// TIA Portal V17 export
// export: Created 2024-09-02T12:50:15.2949432Z, ExportSetting WithDefaults, DisplayName Totally Integrated Automation Portal, DisplayVersion V17, DisplayName TIA Portal Openness, DisplayVersion V17, DisplayName TIA Portal Version Control Interface, DisplayVersion V17, DisplayName STEP 7 Professional, DisplayVersion V17, DisplayName STEP 7 Safety, DisplayVersion V17, DisplayName WinCC Professional, DisplayVersion V17
FUNCTION "AnwFC_ZP_Alarm_OP70" : Void   // FC155, LAD
TITLE = Störmeldungen und Betriebsmeldungen rangieren
{ S7_Optimized_Access := 'TRUE' }
AUTHOR : OlegFuehrus
FAMILY : BA
NAME : BA
VERSION : 0.1
// stored: AutoNumber true, IsIECCheckEnabled false, SetENOAutomatically false, UDAEnableTagReadback false
   VAR_TEMP
      t_bTemp : Bool;
      t_ControlVoltage : Bool;
      t_StartReady : Bool;
      t_OverviewStartCon : Bool;
      t_EStop_NOK : Bool;
      t_Fault : Bool;
      t_oppen_SG : Array[1..8] of Bool;
      t_wert : Byte;
      t_status : Word;
      t_RetValSFC : Int;
      _NumOf_ParFlt_General : Int;
      _NumOf_SQFlt_General : Int;
      _NumOf_Flt_General_A : Int;
      _NumOf_Flt_General_B : Int;
      _NumOf_Flt_SubSys : Int;
      _NumOf_Reports : Int;
      _NumOf_Rep : Int;
   END_VAR
   VAR_TEMP   // added for the SCL form of the ladder/FBD networks
      _w1 : Bool;
      _w2 : Bool;
      _w3 : Bool;
      _w4 : Bool;
      _w5 : Bool;
   END_VAR
BEGIN

REGION Network 1: INIT
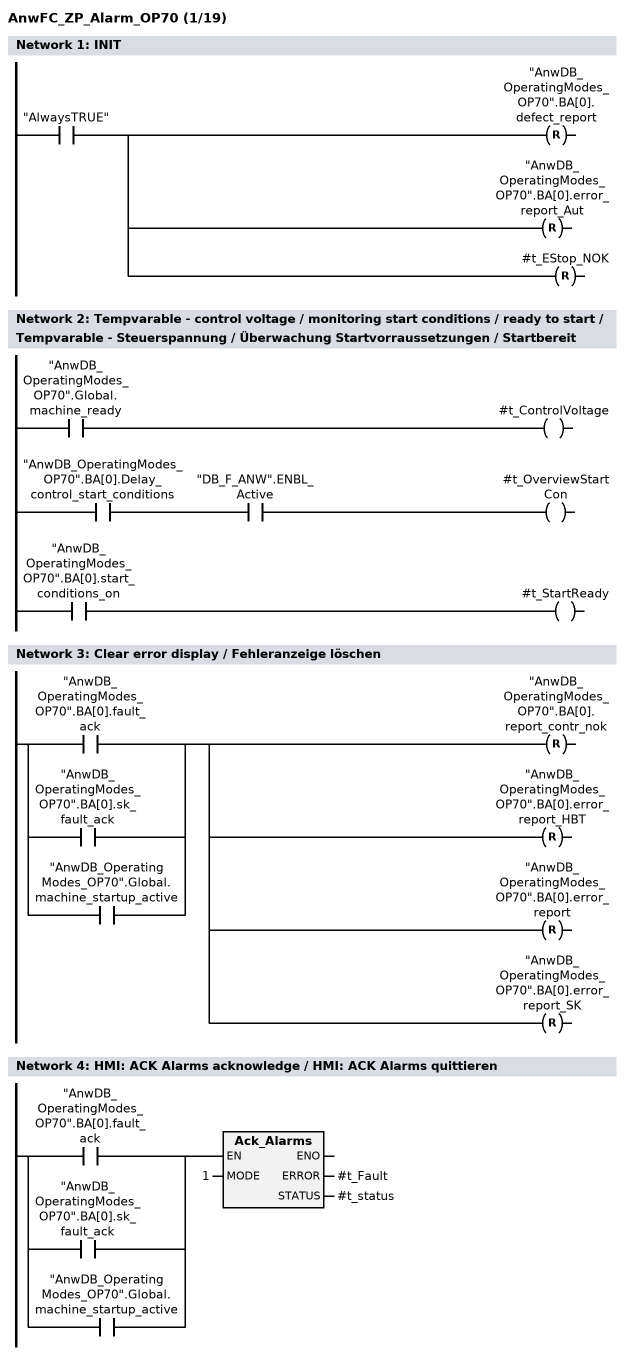
   RUNG wire#powerrail
      Contact( "AlwaysTRUE" )
      wire#w1
      R_Coil( "AnwDB_OperatingModes_OP70".BA[0].defect_report )
   END_RUNG
   RUNG wire#w1
      R_Coil( "AnwDB_OperatingModes_OP70".BA[0].error_report_Aut )
   END_RUNG
   RUNG wire#w1
      R_Coil( #t_EStop_NOK )
   END_RUNG
   // the same network as SCL:
   IF "AlwaysTRUE" THEN
       "AnwDB_OperatingModes_OP70".BA[0].defect_report := FALSE;
       "AnwDB_OperatingModes_OP70".BA[0].error_report_Aut := FALSE;
       #t_EStop_NOK := FALSE;
   END_IF;
END_REGION

REGION Network 2: Tempvarable - control voltage / monitoring start conditions / ready to start / Tempvarable - Steuerspannung / Überwachung Startvorraussetzungen / Startbereit
   RUNG wire#powerrail
      Contact( "AnwDB_OperatingModes_OP70".Global.machine_ready )
      Coil( #t_ControlVoltage )
   END_RUNG
   RUNG wire#powerrail
      Contact( "AnwDB_OperatingModes_OP70".BA[0].Delay_control_start_conditions )
      Contact( "DB_F_ANW".ENBL_Active )
      Coil( #t_OverviewStartCon )
   END_RUNG
   RUNG wire#powerrail
      Contact( "AnwDB_OperatingModes_OP70".BA[0].start_conditions_on )
      Coil( #t_StartReady )
   END_RUNG
   // the same network as SCL:
   #t_ControlVoltage := "AnwDB_OperatingModes_OP70".Global.machine_ready;
   #t_OverviewStartCon := "AnwDB_OperatingModes_OP70".BA[0].Delay_control_start_conditions AND "DB_F_ANW".ENBL_Active;
   #t_StartReady := "AnwDB_OperatingModes_OP70".BA[0].start_conditions_on;
END_REGION

REGION Network 3: Clear error display / Fehleranzeige löschen
   RUNG wire#powerrail
      Contact( "AnwDB_OperatingModes_OP70".BA[0].fault_ack )
      wire#w1
      R_Coil( "AnwDB_OperatingModes_OP70".BA[0].report_contr_nok )
   END_RUNG
   RUNG wire#powerrail
      Contact( "AnwDB_OperatingModes_OP70".BA[0].sk_fault_ack )
   END_RUNG wire#w1
   RUNG wire#powerrail
      Contact( "AnwDB_OperatingModes_OP70".Global.machine_startup_active )
   END_RUNG wire#w1
   RUNG wire#w1
      R_Coil( "AnwDB_OperatingModes_OP70".BA[0].error_report_HBT )
   END_RUNG
   RUNG wire#w1
      R_Coil( "AnwDB_OperatingModes_OP70".BA[0].error_report )
   END_RUNG
   RUNG wire#w1
      R_Coil( "AnwDB_OperatingModes_OP70".BA[0].error_report_SK )
   END_RUNG
   // the same network as SCL:
   #_w1 := "AnwDB_OperatingModes_OP70".BA[0].fault_ack OR "AnwDB_OperatingModes_OP70".BA[0].sk_fault_ack OR "AnwDB_OperatingModes_OP70".Global.machine_startup_active;
   IF #_w1 THEN
       "AnwDB_OperatingModes_OP70".BA[0].report_contr_nok := FALSE;
       "AnwDB_OperatingModes_OP70".BA[0].error_report_HBT := FALSE;
       "AnwDB_OperatingModes_OP70".BA[0].error_report := FALSE;
       "AnwDB_OperatingModes_OP70".BA[0].error_report_SK := FALSE;
   END_IF;
END_REGION

REGION Network 4: HMI: ACK Alarms acknowledge / HMI: ACK Alarms quittieren
   RUNG wire#powerrail
      Contact( "AnwDB_OperatingModes_OP70".BA[0].fault_ack )
      wire#w1
      Ack_Alarms(MODE := 1, ERROR => #t_Fault, STATUS => #t_status)
   END_RUNG
   RUNG wire#powerrail
      Contact( "AnwDB_OperatingModes_OP70".BA[0].sk_fault_ack )
   END_RUNG wire#w1
   RUNG wire#powerrail
      Contact( "AnwDB_OperatingModes_OP70".Global.machine_startup_active )
   END_RUNG wire#w1
   // the same network as SCL:
   IF "AnwDB_OperatingModes_OP70".BA[0].fault_ack OR "AnwDB_OperatingModes_OP70".BA[0].sk_fault_ack OR "AnwDB_OperatingModes_OP70".Global.machine_startup_active THEN
       Ack_Alarms(MODE := 1, ERROR => #t_Fault, STATUS => #t_status);
   END_IF;
END_REGION

REGION Network 5: Acknowledge fault at MP / Störung am MP quittieren
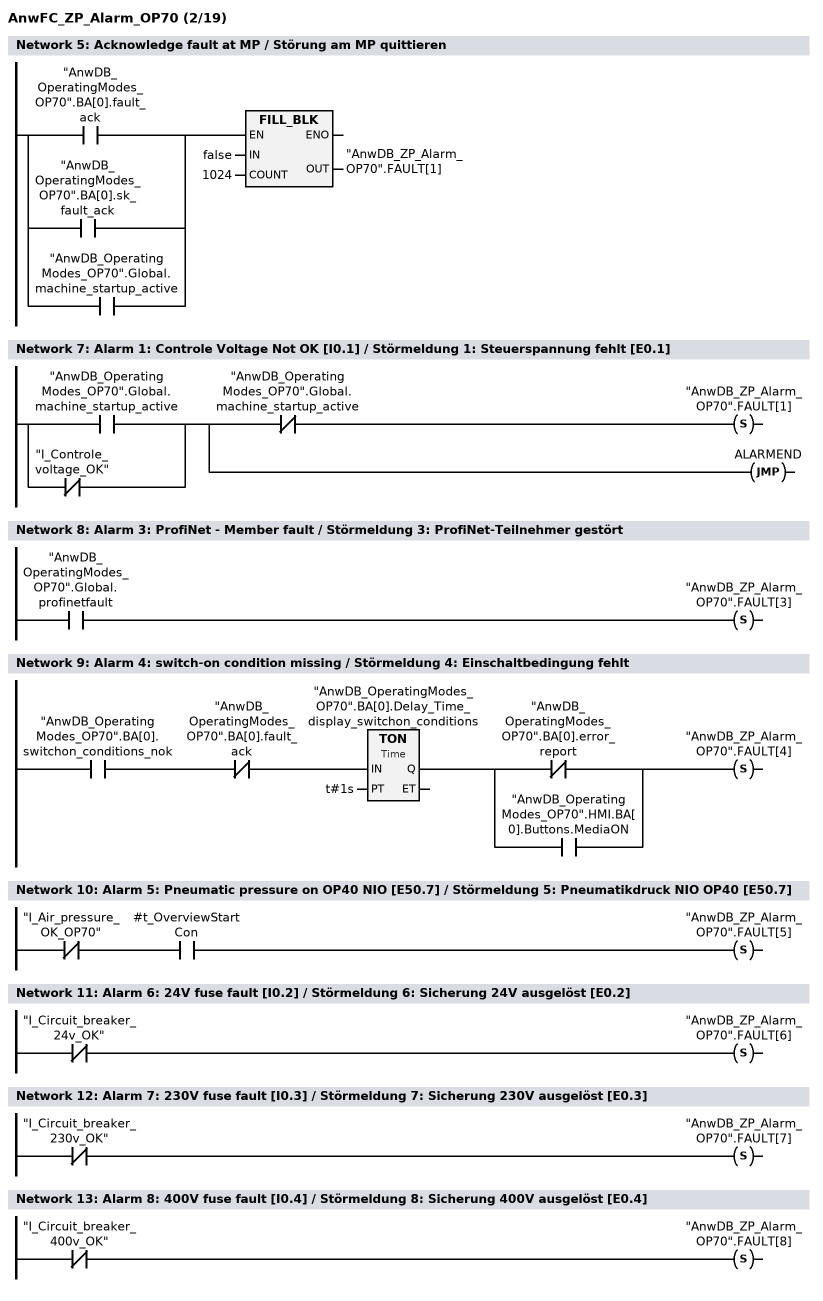
   RUNG wire#powerrail
      Contact( "AnwDB_OperatingModes_OP70".BA[0].fault_ack )
      wire#w1
      FillBlockI(in := false, count := 1024, out => "AnwDB_ZP_Alarm_OP70".FAULT[1])
   END_RUNG
   RUNG wire#powerrail
      Contact( "AnwDB_OperatingModes_OP70".BA[0].sk_fault_ack )
   END_RUNG wire#w1
   RUNG wire#powerrail
      Contact( "AnwDB_OperatingModes_OP70".Global.machine_startup_active )
   END_RUNG wire#w1
   // the same network as SCL:
   IF "AnwDB_OperatingModes_OP70".BA[0].fault_ack OR "AnwDB_OperatingModes_OP70".BA[0].sk_fault_ack OR "AnwDB_OperatingModes_OP70".Global.machine_startup_active THEN
       FILL_BLK(IN := false, COUNT := 1024, OUT => "AnwDB_ZP_Alarm_OP70".FAULT[1]);
   END_IF;
END_REGION

REGION Network 6: ########################### Global Power condition############################### / ########################### Störmeldungen ###############################
END_REGION

REGION Network 7: Alarm 1: Controle Voltage Not OK [I0.1] / Störmeldung 1: Steuerspannung fehlt [E0.1]
   RUNG wire#powerrail
      Contact( "AnwDB_OperatingModes_OP70".Global.machine_startup_active )
      wire#w1
      I_Contact( "AnwDB_OperatingModes_OP70".Global.machine_startup_active )
      S_Coil( "AnwDB_ZP_Alarm_OP70".FAULT[1] )
   END_RUNG
   RUNG wire#powerrail
      I_Contact( "I_Controle_voltage_OK" )
   END_RUNG wire#w1
   RUNG wire#w1
      JumpCoil( ALARMEND )
   END_RUNG
   // the same network as SCL:
   #_w1 := "AnwDB_OperatingModes_OP70".Global.machine_startup_active OR NOT "I_Controle_voltage_OK";
   IF #_w1 AND NOT "AnwDB_OperatingModes_OP70".Global.machine_startup_active THEN
       "AnwDB_ZP_Alarm_OP70".FAULT[1] := TRUE;
   END_IF;
   IF #_w1 THEN GOTO ALARMEND; END_IF;
END_REGION

REGION Network 8: Alarm 3: ProfiNet - Member fault / Störmeldung 3: ProfiNet-Teilnehmer gestört
   RUNG wire#powerrail
      Contact( "AnwDB_OperatingModes_OP70".Global.profinetfault )
      S_Coil( "AnwDB_ZP_Alarm_OP70".FAULT[3] )
   END_RUNG
   // the same network as SCL:
   IF "AnwDB_OperatingModes_OP70".Global.profinetfault THEN "AnwDB_ZP_Alarm_OP70".FAULT[3] := TRUE; END_IF;
END_REGION

REGION Network 9: Alarm 4: switch-on condition missing / Störmeldung 4: Einschaltbedingung fehlt
   RUNG wire#powerrail
      Contact( "AnwDB_OperatingModes_OP70".BA[0].switchon_conditions_nok )
      I_Contact( "AnwDB_OperatingModes_OP70".BA[0].fault_ack )
      { S7_Templates := "time_type := Time" } "AnwDB_OperatingModes_OP70".BA[0].Delay_Time_display_switchon_conditions.TON(pt := t#1s, et =>)
      wire#w1
      I_Contact( "AnwDB_OperatingModes_OP70".BA[0].error_report )
      wire#w2
      S_Coil( "AnwDB_ZP_Alarm_OP70".FAULT[4] )
   END_RUNG
   RUNG wire#w1
      Contact( "AnwDB_OperatingModes_OP70".HMI.BA[0].Buttons.MediaON )
   END_RUNG wire#w2
   // the same network as SCL:
   "AnwDB_OperatingModes_OP70".BA[0].Delay_Time_display_switchon_conditions.TON(IN := "AnwDB_OperatingModes_OP70".BA[0].switchon_conditions_nok AND NOT "AnwDB_OperatingModes_OP70".BA[0].fault_ack,
                           PT := t#1s);
   IF "AnwDB_OperatingModes_OP70".BA[0].Delay_Time_display_switchon_conditions.Q AND (NOT "AnwDB_OperatingModes_OP70".BA[0].error_report OR "AnwDB_OperatingModes_OP70".HMI.BA[0].Buttons.MediaON) THEN
       "AnwDB_ZP_Alarm_OP70".FAULT[4] := TRUE;
   END_IF;
END_REGION

REGION Network 10: Alarm 5: Pneumatic pressure on OP40 NIO [E50.7] / Störmeldung 5: Pneumatikdruck NIO OP40 [E50.7]
   RUNG wire#powerrail
      I_Contact( "I_Air_pressure_OK_OP70" )
      Contact( #t_OverviewStartCon )
      S_Coil( "AnwDB_ZP_Alarm_OP70".FAULT[5] )
   END_RUNG
   // the same network as SCL:
   IF NOT "I_Air_pressure_OK_OP70" AND #t_OverviewStartCon THEN
       "AnwDB_ZP_Alarm_OP70".FAULT[5] := TRUE;
   END_IF;
END_REGION

REGION Network 11: Alarm 6: 24V fuse fault [I0.2] / Störmeldung 6: Sicherung 24V ausgelöst [E0.2]
   RUNG wire#powerrail
      I_Contact( "I_Circuit_breaker_24v_OK" )
      S_Coil( "AnwDB_ZP_Alarm_OP70".FAULT[6] )
   END_RUNG
   // the same network as SCL:
   IF NOT "I_Circuit_breaker_24v_OK" THEN "AnwDB_ZP_Alarm_OP70".FAULT[6] := TRUE; END_IF;
END_REGION

REGION Network 12: Alarm 7: 230V fuse fault [I0.3] / Störmeldung 7: Sicherung 230V ausgelöst [E0.3]
   RUNG wire#powerrail
      I_Contact( "I_Circuit_breaker_230v_OK" )
      S_Coil( "AnwDB_ZP_Alarm_OP70".FAULT[7] )
   END_RUNG
   // the same network as SCL:
   IF NOT "I_Circuit_breaker_230v_OK" THEN "AnwDB_ZP_Alarm_OP70".FAULT[7] := TRUE; END_IF;
END_REGION

REGION Network 13: Alarm 8: 400V fuse fault [I0.4] / Störmeldung 8: Sicherung 400V ausgelöst [E0.4]
   RUNG wire#powerrail
      I_Contact( "I_Circuit_breaker_400v_OK" )
      S_Coil( "AnwDB_ZP_Alarm_OP70".FAULT[8] )
   END_RUNG
   // the same network as SCL:
   IF NOT "I_Circuit_breaker_400v_OK" THEN "AnwDB_ZP_Alarm_OP70".FAULT[8] := TRUE; END_IF;
END_REGION

REGION Network 14: Power Condition: ENDE ########################## / ESB: ENDE ##########################
END_REGION

REGION Network 15: Alarm 25: Reworking in Station / Störmeldung 25: Nacharbeit in Station
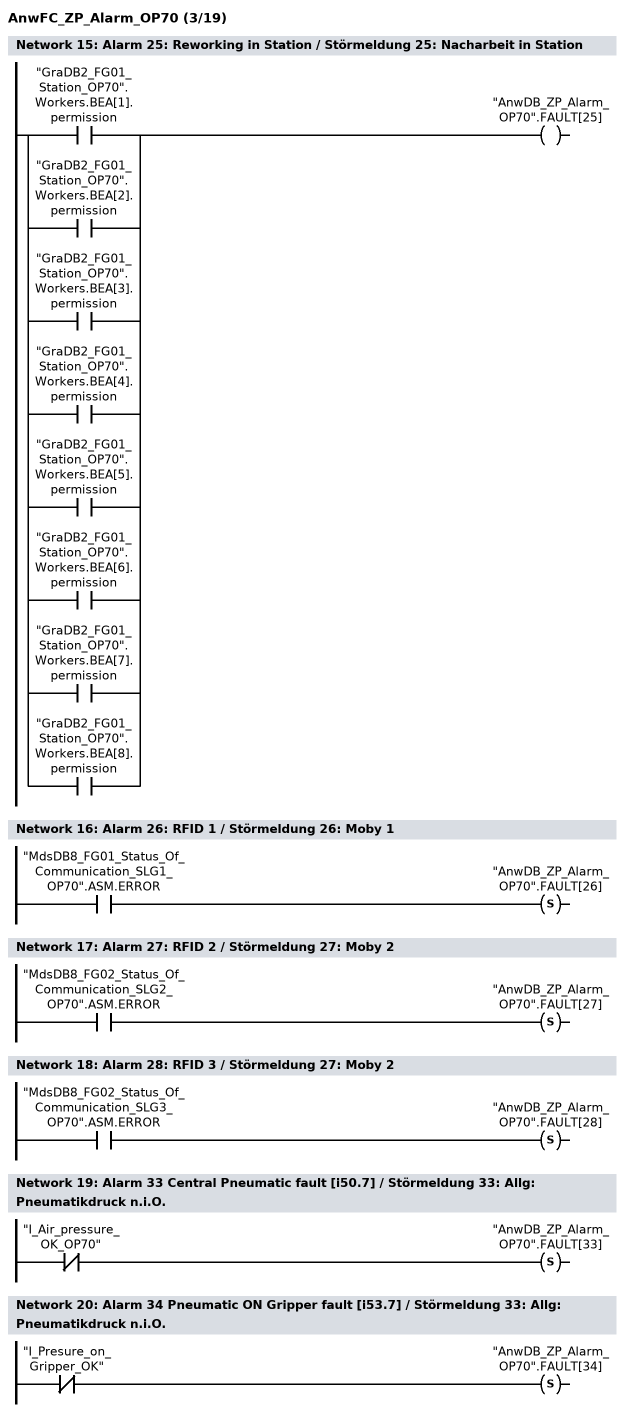
   RUNG wire#powerrail
      Contact( "GraDB2_FG01_Station_OP70".Workers.BEA[1].permission )
      wire#w1
      Coil( "AnwDB_ZP_Alarm_OP70".FAULT[25] )
   END_RUNG
   RUNG wire#powerrail
      Contact( "GraDB2_FG01_Station_OP70".Workers.BEA[2].permission )
   END_RUNG wire#w1
   RUNG wire#powerrail
      Contact( "GraDB2_FG01_Station_OP70".Workers.BEA[3].permission )
   END_RUNG wire#w1
   RUNG wire#powerrail
      Contact( "GraDB2_FG01_Station_OP70".Workers.BEA[4].permission )
   END_RUNG wire#w1
   RUNG wire#powerrail
      Contact( "GraDB2_FG01_Station_OP70".Workers.BEA[5].permission )
   END_RUNG wire#w1
   RUNG wire#powerrail
      Contact( "GraDB2_FG01_Station_OP70".Workers.BEA[6].permission )
   END_RUNG wire#w1
   RUNG wire#powerrail
      Contact( "GraDB2_FG01_Station_OP70".Workers.BEA[7].permission )
   END_RUNG wire#w1
   RUNG wire#powerrail
      Contact( "GraDB2_FG01_Station_OP70".Workers.BEA[8].permission )
   END_RUNG wire#w1
   // the same network as SCL:
   "AnwDB_ZP_Alarm_OP70".FAULT[25] := "GraDB2_FG01_Station_OP70".Workers.BEA[1].permission OR "GraDB2_FG01_Station_OP70".Workers.BEA[2].permission OR "GraDB2_FG01_Station_OP70".Workers.BEA[3].permission OR "GraDB2_FG01_Station_OP70".Workers.BEA[4].permission OR "GraDB2_FG01_Station_OP70".Workers.BEA[5].permission OR "GraDB2_FG01_Station_OP70".Workers.BEA[6].permission OR "GraDB2_FG01_Station_OP70".Workers.BEA[7].permission OR "GraDB2_FG01_Station_OP70".Workers.BEA[8].permission;
END_REGION

REGION Network 16: Alarm 26: RFID 1 / Störmeldung 26: Moby 1
   RUNG wire#powerrail
      Contact( "MdsDB8_FG01_Status_Of_Communication_SLG1_OP70".ASM.ERROR )
      S_Coil( "AnwDB_ZP_Alarm_OP70".FAULT[26] )
   END_RUNG
   // the same network as SCL:
   IF "MdsDB8_FG01_Status_Of_Communication_SLG1_OP70".ASM.ERROR THEN
       "AnwDB_ZP_Alarm_OP70".FAULT[26] := TRUE;
   END_IF;
END_REGION

REGION Network 17: Alarm 27: RFID 2 / Störmeldung 27: Moby 2
   RUNG wire#powerrail
      Contact( "MdsDB8_FG02_Status_Of_Communication_SLG2_OP70".ASM.ERROR )
      S_Coil( "AnwDB_ZP_Alarm_OP70".FAULT[27] )
   END_RUNG
   // the same network as SCL:
   IF "MdsDB8_FG02_Status_Of_Communication_SLG2_OP70".ASM.ERROR THEN
       "AnwDB_ZP_Alarm_OP70".FAULT[27] := TRUE;
   END_IF;
END_REGION

REGION Network 18: Alarm 28: RFID 3 / Störmeldung 27: Moby 2
   RUNG wire#powerrail
      Contact( "MdsDB8_FG02_Status_Of_Communication_SLG3_OP70".ASM.ERROR )
      S_Coil( "AnwDB_ZP_Alarm_OP70".FAULT[28] )
   END_RUNG
   // the same network as SCL:
   IF "MdsDB8_FG02_Status_Of_Communication_SLG3_OP70".ASM.ERROR THEN
       "AnwDB_ZP_Alarm_OP70".FAULT[28] := TRUE;
   END_IF;
END_REGION

REGION Network 19: Alarm 33 Central Pneumatic fault [i50.7] / Störmeldung 33: Allg: Pneumatikdruck n.i.O.
   RUNG wire#powerrail
      I_Contact( "I_Air_pressure_OK_OP70" )
      S_Coil( "AnwDB_ZP_Alarm_OP70".FAULT[33] )
   END_RUNG
   // the same network as SCL:
   IF NOT "I_Air_pressure_OK_OP70" THEN "AnwDB_ZP_Alarm_OP70".FAULT[33] := TRUE; END_IF;
END_REGION

REGION Network 20: Alarm 34 Pneumatic ON Gripper fault [i53.7] / Störmeldung 33: Allg: Pneumatikdruck n.i.O.
   RUNG wire#powerrail
      I_Contact( "I_Presure_on_Gripper_OK" )
      S_Coil( "AnwDB_ZP_Alarm_OP70".FAULT[34] )
   END_RUNG
   // the same network as SCL:
   IF NOT "I_Presure_on_Gripper_OK" THEN "AnwDB_ZP_Alarm_OP70".FAULT[34] := TRUE; END_IF;
END_REGION

REGION Network 21: Alarm 42: Control cabinet temperature exceeded (> 30 minutes) [E0.7] / Störmeldung 42: Temperatur Schaltschrank überschritten (>30 Minuten) [E0.7]
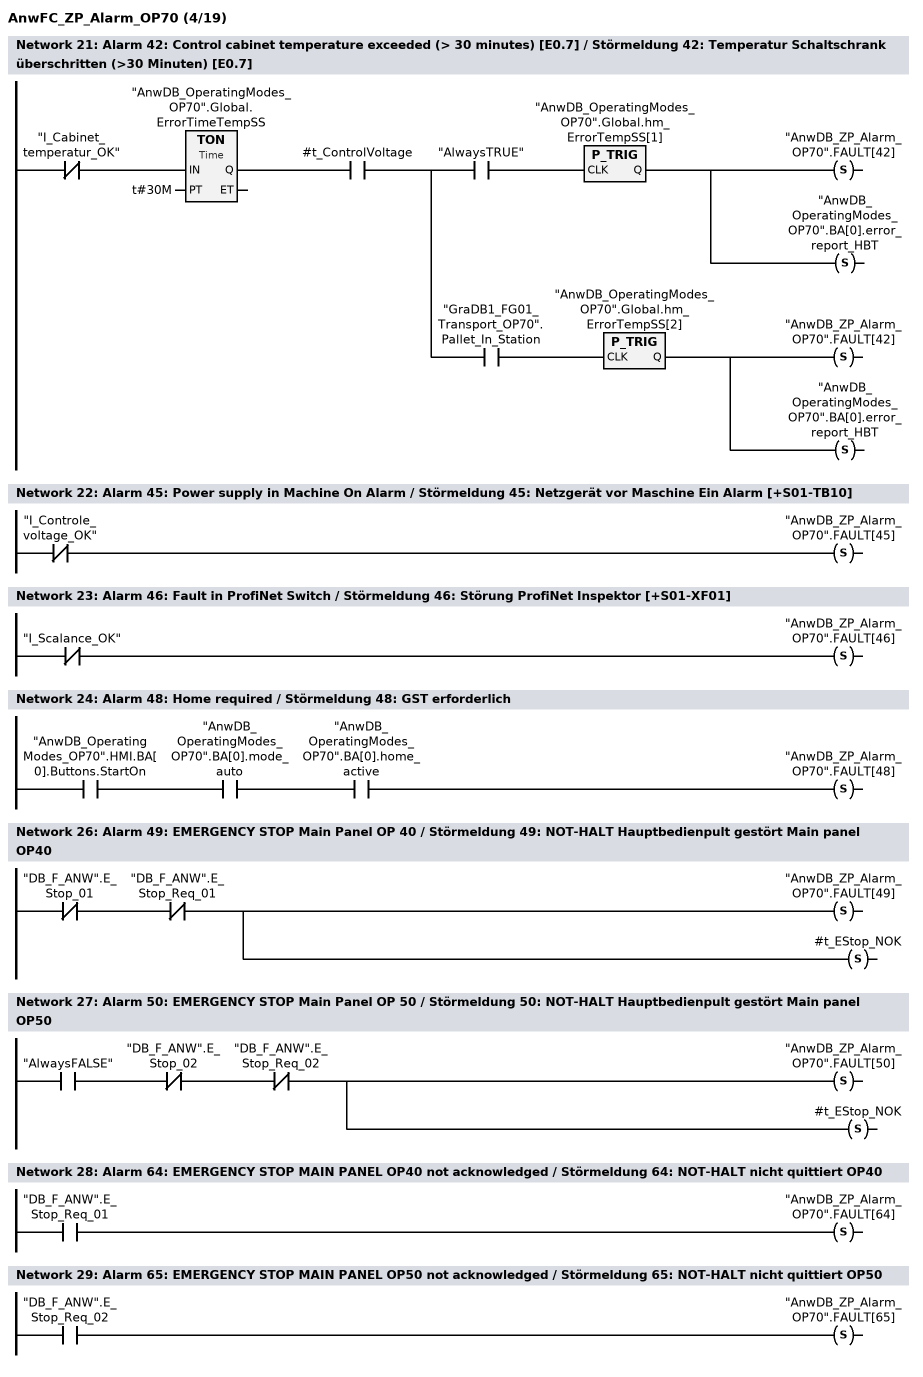
   RUNG wire#powerrail
      I_Contact( "I_Cabinet_temperatur_OK" )
      { S7_Templates := "time_type := Time" } "AnwDB_OperatingModes_OP70".Global.ErrorTimeTempSS.TON(pt := t#30M, et =>)
      Contact( #t_ControlVoltage )
      wire#w1
      Contact( "AlwaysTRUE" )
      P_Trig( "AnwDB_OperatingModes_OP70".Global.hm_ErrorTempSS[1] )
      wire#w2
      S_Coil( "AnwDB_ZP_Alarm_OP70".FAULT[42] )
   END_RUNG
   RUNG wire#w2
      S_Coil( "AnwDB_OperatingModes_OP70".BA[0].error_report_HBT )
   END_RUNG
   RUNG wire#w1
      Contact( "GraDB1_FG01_Transport_OP70".Pallet_In_Station )
      P_Trig( "AnwDB_OperatingModes_OP70".Global.hm_ErrorTempSS[2] )
      wire#w3
      S_Coil( "AnwDB_ZP_Alarm_OP70".FAULT[42] )
   END_RUNG
   RUNG wire#w3
      S_Coil( "AnwDB_OperatingModes_OP70".BA[0].error_report_HBT )
   END_RUNG
   // the same network as SCL:
   "AnwDB_OperatingModes_OP70".Global.ErrorTimeTempSS.TON(IN := NOT "I_Cabinet_temperatur_OK", PT := t#30M);
   #_w1 := "AnwDB_OperatingModes_OP70".Global.ErrorTimeTempSS.Q AND #t_ControlVoltage;
   #_w2 := #_w1 AND "AlwaysTRUE";
   #_w3 := #_w2 AND NOT "AnwDB_OperatingModes_OP70".Global.hm_ErrorTempSS[1];   // rising edge
   "AnwDB_OperatingModes_OP70".Global.hm_ErrorTempSS[1] := #_w2;
   IF #_w3 THEN
       "AnwDB_ZP_Alarm_OP70".FAULT[42] := TRUE;
       "AnwDB_OperatingModes_OP70".BA[0].error_report_HBT := TRUE;
   END_IF;
   #_w4 := #_w1 AND "GraDB1_FG01_Transport_OP70".Pallet_In_Station;
   #_w5 := #_w4 AND NOT "AnwDB_OperatingModes_OP70".Global.hm_ErrorTempSS[2];   // rising edge
   "AnwDB_OperatingModes_OP70".Global.hm_ErrorTempSS[2] := #_w4;
   IF #_w5 THEN
       "AnwDB_ZP_Alarm_OP70".FAULT[42] := TRUE;
       "AnwDB_OperatingModes_OP70".BA[0].error_report_HBT := TRUE;
   END_IF;
END_REGION

REGION Network 22: Alarm 45: Power supply in Machine On Alarm / Störmeldung 45: Netzgerät vor Maschine Ein Alarm [+S01-TB10]
   RUNG wire#powerrail
      I_Contact( "I_Controle_voltage_OK" )
      S_Coil( "AnwDB_ZP_Alarm_OP70".FAULT[45] )
   END_RUNG
   // the same network as SCL:
   IF NOT "I_Controle_voltage_OK" THEN "AnwDB_ZP_Alarm_OP70".FAULT[45] := TRUE; END_IF;
END_REGION

REGION Network 23: Alarm 46: Fault in ProfiNet Switch / Störmeldung 46: Störung ProfiNet Inspektor [+S01-XF01]
   RUNG wire#powerrail
      I_Contact( "I_Scalance_OK" )
      S_Coil( "AnwDB_ZP_Alarm_OP70".FAULT[46] )
   END_RUNG
   // the same network as SCL:
   IF NOT "I_Scalance_OK" THEN "AnwDB_ZP_Alarm_OP70".FAULT[46] := TRUE; END_IF;
END_REGION

REGION Network 24: Alarm 48: Home required / Störmeldung 48: GST erforderlich
   RUNG wire#powerrail
      Contact( "AnwDB_OperatingModes_OP70".HMI.BA[0].Buttons.StartOn )
      Contact( "AnwDB_OperatingModes_OP70".BA[0].mode_auto )
      Contact( "AnwDB_OperatingModes_OP70".BA[0].home_active )
      S_Coil( "AnwDB_ZP_Alarm_OP70".FAULT[48] )
   END_RUNG
   // the same network as SCL:
   IF "AnwDB_OperatingModes_OP70".HMI.BA[0].Buttons.StartOn AND "AnwDB_OperatingModes_OP70".BA[0].mode_auto AND "AnwDB_OperatingModes_OP70".BA[0].home_active THEN
       "AnwDB_ZP_Alarm_OP70".FAULT[48] := TRUE;
   END_IF;
END_REGION

REGION Network 25: Allg: ENDE ############################
END_REGION

REGION Network 26: Alarm 49: EMERGENCY STOP Main Panel OP 40 / Störmeldung 49: NOT-HALT Hauptbedienpult gestört Main panel OP40
   RUNG wire#powerrail
      I_Contact( "DB_F_ANW".E_Stop_01 )
      I_Contact( "DB_F_ANW".E_Stop_Req_01 )
      wire#w1
      S_Coil( "AnwDB_ZP_Alarm_OP70".FAULT[49] )
   END_RUNG
   RUNG wire#w1
      S_Coil( #t_EStop_NOK )
   END_RUNG
   // the same network as SCL:
   IF NOT "DB_F_ANW".E_Stop_01 AND NOT "DB_F_ANW".E_Stop_Req_01 THEN
       "AnwDB_ZP_Alarm_OP70".FAULT[49] := TRUE;
       #t_EStop_NOK := TRUE;
   END_IF;
END_REGION

REGION Network 27: Alarm 50: EMERGENCY STOP Main Panel OP 50 / Störmeldung 50: NOT-HALT Hauptbedienpult gestört Main panel OP50
   RUNG wire#powerrail
      Contact( "AlwaysFALSE" )
      I_Contact( "DB_F_ANW".E_Stop_02 )
      I_Contact( "DB_F_ANW".E_Stop_Req_02 )
      wire#w1
      S_Coil( "AnwDB_ZP_Alarm_OP70".FAULT[50] )
   END_RUNG
   RUNG wire#w1
      S_Coil( #t_EStop_NOK )
   END_RUNG
   // the same network as SCL:
   IF "AlwaysFALSE" AND NOT "DB_F_ANW".E_Stop_02 AND NOT "DB_F_ANW".E_Stop_Req_02 THEN
       "AnwDB_ZP_Alarm_OP70".FAULT[50] := TRUE;
       #t_EStop_NOK := TRUE;
   END_IF;
END_REGION

REGION Network 28: Alarm 64: EMERGENCY STOP MAIN PANEL OP40 not acknowledged / Störmeldung 64: NOT-HALT nicht quittiert OP40
   RUNG wire#powerrail
      Contact( "DB_F_ANW".E_Stop_Req_01 )
      S_Coil( "AnwDB_ZP_Alarm_OP70".FAULT[64] )
   END_RUNG
   // the same network as SCL:
   IF "DB_F_ANW".E_Stop_Req_01 THEN "AnwDB_ZP_Alarm_OP70".FAULT[64] := TRUE; END_IF;
END_REGION

REGION Network 29: Alarm 65: EMERGENCY STOP MAIN PANEL OP50 not acknowledged / Störmeldung 65: NOT-HALT nicht quittiert OP50
   RUNG wire#powerrail
      Contact( "DB_F_ANW".E_Stop_Req_02 )
      S_Coil( "AnwDB_ZP_Alarm_OP70".FAULT[65] )
   END_RUNG
   // the same network as SCL:
   IF "DB_F_ANW".E_Stop_Req_02 THEN "AnwDB_ZP_Alarm_OP70".FAULT[65] := TRUE; END_IF;
END_REGION

REGION Network 30: Alarm 66: Safety Door opened / Störmeldung 66: Schutztür 1 offen
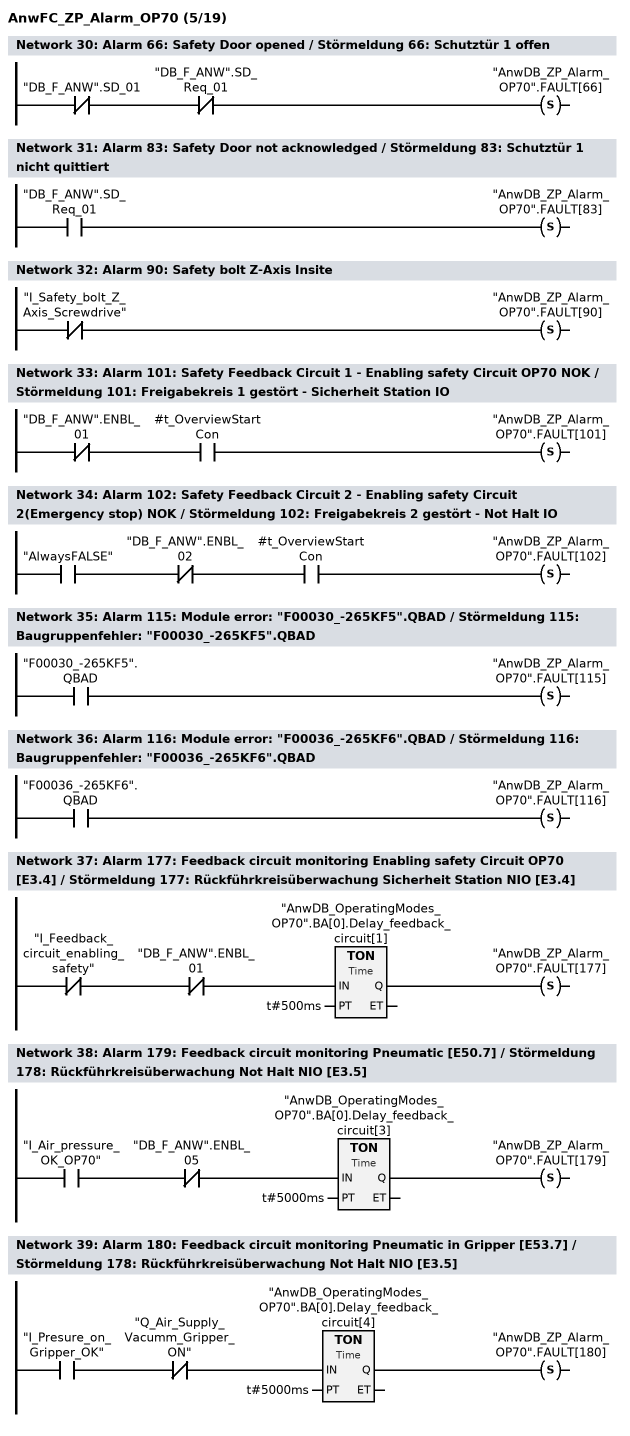
   RUNG wire#powerrail
      I_Contact( "DB_F_ANW".SD_01 )
      I_Contact( "DB_F_ANW".SD_Req_01 )
      S_Coil( "AnwDB_ZP_Alarm_OP70".FAULT[66] )
   END_RUNG
   // the same network as SCL:
   IF NOT "DB_F_ANW".SD_01 AND NOT "DB_F_ANW".SD_Req_01 THEN "AnwDB_ZP_Alarm_OP70".FAULT[66] := TRUE; END_IF;
END_REGION

REGION Network 31: Alarm 83: Safety Door not acknowledged / Störmeldung 83: Schutztür 1 nicht quittiert
   RUNG wire#powerrail
      Contact( "DB_F_ANW".SD_Req_01 )
      S_Coil( "AnwDB_ZP_Alarm_OP70".FAULT[83] )
   END_RUNG
   // the same network as SCL:
   IF "DB_F_ANW".SD_Req_01 THEN "AnwDB_ZP_Alarm_OP70".FAULT[83] := TRUE; END_IF;
END_REGION

REGION Network 32: Alarm 90: Safety bolt Z-Axis Insite
   RUNG wire#powerrail
      I_Contact( "I_Safety_bolt_Z_Axis_Screwdrive" )
      S_Coil( "AnwDB_ZP_Alarm_OP70".FAULT[90] )
   END_RUNG
   // the same network as SCL:
   IF NOT "I_Safety_bolt_Z_Axis_Screwdrive" THEN "AnwDB_ZP_Alarm_OP70".FAULT[90] := TRUE; END_IF;
END_REGION

REGION Network 33: Alarm 101: Safety Feedback Circuit 1 - Enabling safety Circuit OP70 NOK / Störmeldung 101: Freigabekreis 1 gestört - Sicherheit Station IO
   RUNG wire#powerrail
      I_Contact( "DB_F_ANW".ENBL_01 )
      Contact( #t_OverviewStartCon )
      S_Coil( "AnwDB_ZP_Alarm_OP70".FAULT[101] )
   END_RUNG
   // the same network as SCL:
   IF NOT "DB_F_ANW".ENBL_01 AND #t_OverviewStartCon THEN "AnwDB_ZP_Alarm_OP70".FAULT[101] := TRUE; END_IF;
END_REGION

REGION Network 34: Alarm 102: Safety Feedback Circuit 2 - Enabling safety Circuit 2(Emergency stop) NOK / Störmeldung 102: Freigabekreis 2 gestört - Not Halt IO
   RUNG wire#powerrail
      Contact( "AlwaysFALSE" )
      I_Contact( "DB_F_ANW".ENBL_02 )
      Contact( #t_OverviewStartCon )
      S_Coil( "AnwDB_ZP_Alarm_OP70".FAULT[102] )
   END_RUNG
   // the same network as SCL:
   IF "AlwaysFALSE" AND NOT "DB_F_ANW".ENBL_02 AND #t_OverviewStartCon THEN
       "AnwDB_ZP_Alarm_OP70".FAULT[102] := TRUE;
   END_IF;
END_REGION

REGION Network 35: Alarm 115: Module error: "F00030_-265KF5".QBAD / Störmeldung 115: Baugruppenfehler: "F00030_-265KF5".QBAD
   RUNG wire#powerrail
      Contact( "F00030_-265KF5".QBAD )
      S_Coil( "AnwDB_ZP_Alarm_OP70".FAULT[115] )
   END_RUNG
   // the same network as SCL:
   IF "F00030_-265KF5".QBAD THEN "AnwDB_ZP_Alarm_OP70".FAULT[115] := TRUE; END_IF;
END_REGION

REGION Network 36: Alarm 116: Module error: "F00036_-265KF6".QBAD / Störmeldung 116: Baugruppenfehler: "F00036_-265KF6".QBAD
   RUNG wire#powerrail
      Contact( "F00036_-265KF6".QBAD )
      S_Coil( "AnwDB_ZP_Alarm_OP70".FAULT[116] )
   END_RUNG
   // the same network as SCL:
   IF "F00036_-265KF6".QBAD THEN "AnwDB_ZP_Alarm_OP70".FAULT[116] := TRUE; END_IF;
END_REGION

REGION Network 37: Alarm 177: Feedback circuit monitoring Enabling safety Circuit OP70 [E3.4] / Störmeldung 177: Rückführkreisüberwachung Sicherheit Station NIO [E3.4]
   RUNG wire#powerrail
      I_Contact( "I_Feedback_circuit_enabling_safety" )
      I_Contact( "DB_F_ANW".ENBL_01 )
      { S7_Templates := "time_type := Time" } "AnwDB_OperatingModes_OP70".BA[0].Delay_feedback_circuit[1].TON(pt := t#500ms, et =>)
      S_Coil( "AnwDB_ZP_Alarm_OP70".FAULT[177] )
   END_RUNG
   // the same network as SCL:
   "AnwDB_OperatingModes_OP70".BA[0].Delay_feedback_circuit[1].TON(IN := NOT "I_Feedback_circuit_enabling_safety" AND NOT "DB_F_ANW".ENBL_01,
                           PT := t#500ms);
   IF "AnwDB_OperatingModes_OP70".BA[0].Delay_feedback_circuit[1].Q THEN
       "AnwDB_ZP_Alarm_OP70".FAULT[177] := TRUE;
   END_IF;
END_REGION

REGION Network 38: Alarm 179: Feedback circuit monitoring Pneumatic [E50.7] / Störmeldung 178: Rückführkreisüberwachung Not Halt NIO [E3.5]
   RUNG wire#powerrail
      Contact( "I_Air_pressure_OK_OP70" )
      I_Contact( "DB_F_ANW".ENBL_05 )
      { S7_Templates := "time_type := Time" } "AnwDB_OperatingModes_OP70".BA[0].Delay_feedback_circuit[3].TON(pt := t#5000ms, et =>)
      S_Coil( "AnwDB_ZP_Alarm_OP70".FAULT[179] )
   END_RUNG
   // the same network as SCL:
   "AnwDB_OperatingModes_OP70".BA[0].Delay_feedback_circuit[3].TON(IN := "I_Air_pressure_OK_OP70" AND NOT "DB_F_ANW".ENBL_05,
                           PT := t#5000ms);
   IF "AnwDB_OperatingModes_OP70".BA[0].Delay_feedback_circuit[3].Q THEN
       "AnwDB_ZP_Alarm_OP70".FAULT[179] := TRUE;
   END_IF;
END_REGION

REGION Network 39: Alarm 180: Feedback circuit monitoring Pneumatic in Gripper [E53.7] / Störmeldung 178: Rückführkreisüberwachung Not Halt NIO [E3.5]
   RUNG wire#powerrail
      Contact( "I_Presure_on_Gripper_OK" )
      I_Contact( "Q_Air_Supply_Vacumm_Gripper_ON" )
      { S7_Templates := "time_type := Time" } "AnwDB_OperatingModes_OP70".BA[0].Delay_feedback_circuit[4].TON(pt := t#5000ms, et =>)
      S_Coil( "AnwDB_ZP_Alarm_OP70".FAULT[180] )
   END_RUNG
   // the same network as SCL:
   "AnwDB_OperatingModes_OP70".BA[0].Delay_feedback_circuit[4].TON(IN := "I_Presure_on_Gripper_OK" AND NOT "Q_Air_Supply_Vacumm_Gripper_ON",
                           PT := t#5000ms);
   IF "AnwDB_OperatingModes_OP70".BA[0].Delay_feedback_circuit[4].Q THEN
       "AnwDB_ZP_Alarm_OP70".FAULT[180] := TRUE;
   END_IF;
END_REGION

REGION Network 40: Alarm 265: Feedback - Power on external device controle [ixxxx] / Störmeldung 265: Schütz
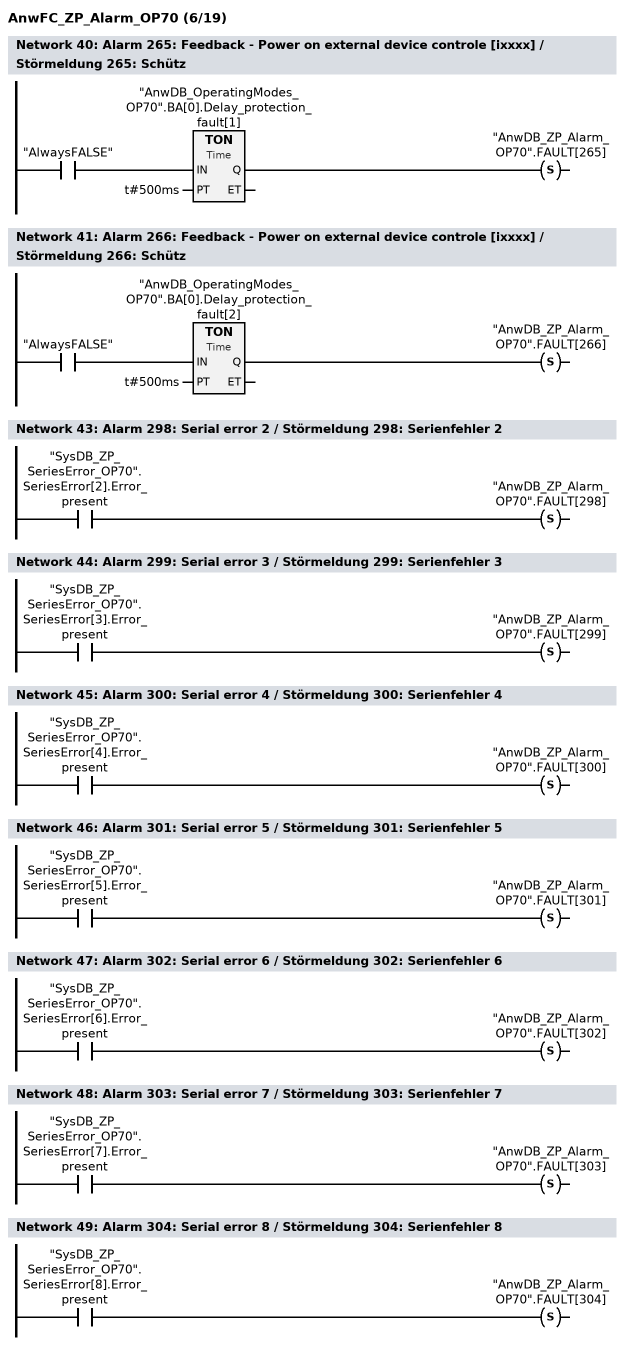
   RUNG wire#powerrail
      Contact( "AlwaysFALSE" )
      { S7_Templates := "time_type := Time" } "AnwDB_OperatingModes_OP70".BA[0].Delay_protection_fault[1].TON(pt := t#500ms, et =>)
      S_Coil( "AnwDB_ZP_Alarm_OP70".FAULT[265] )
   END_RUNG
   // the same network as SCL:
   "AnwDB_OperatingModes_OP70".BA[0].Delay_protection_fault[1].TON(IN := "AlwaysFALSE", PT := t#500ms);
   IF "AnwDB_OperatingModes_OP70".BA[0].Delay_protection_fault[1].Q THEN
       "AnwDB_ZP_Alarm_OP70".FAULT[265] := TRUE;
   END_IF;
END_REGION

REGION Network 41: Alarm 266: Feedback - Power on external device controle [ixxxx] / Störmeldung 266: Schütz
   RUNG wire#powerrail
      Contact( "AlwaysFALSE" )
      { S7_Templates := "time_type := Time" } "AnwDB_OperatingModes_OP70".BA[0].Delay_protection_fault[2].TON(pt := t#500ms, et =>)
      S_Coil( "AnwDB_ZP_Alarm_OP70".FAULT[266] )
   END_RUNG
   // the same network as SCL:
   "AnwDB_OperatingModes_OP70".BA[0].Delay_protection_fault[2].TON(IN := "AlwaysFALSE", PT := t#500ms);
   IF "AnwDB_OperatingModes_OP70".BA[0].Delay_protection_fault[2].Q THEN
       "AnwDB_ZP_Alarm_OP70".FAULT[266] := TRUE;
   END_IF;
END_REGION

REGION Network 42: Alarm 297:Serial error 1 / Störmeldung 297: Serienfehler 1
END_REGION

REGION Network 43: Alarm 298: Serial error 2 / Störmeldung 298: Serienfehler 2
   RUNG wire#powerrail
      Contact( "SysDB_ZP_SeriesError_OP70".SeriesError[2].Error_present )
      S_Coil( "AnwDB_ZP_Alarm_OP70".FAULT[298] )
   END_RUNG
   // the same network as SCL:
   IF "SysDB_ZP_SeriesError_OP70".SeriesError[2].Error_present THEN
       "AnwDB_ZP_Alarm_OP70".FAULT[298] := TRUE;
   END_IF;
END_REGION

REGION Network 44: Alarm 299: Serial error 3 / Störmeldung 299: Serienfehler 3
   RUNG wire#powerrail
      Contact( "SysDB_ZP_SeriesError_OP70".SeriesError[3].Error_present )
      S_Coil( "AnwDB_ZP_Alarm_OP70".FAULT[299] )
   END_RUNG
   // the same network as SCL:
   IF "SysDB_ZP_SeriesError_OP70".SeriesError[3].Error_present THEN
       "AnwDB_ZP_Alarm_OP70".FAULT[299] := TRUE;
   END_IF;
END_REGION

REGION Network 45: Alarm 300: Serial error 4 / Störmeldung 300: Serienfehler 4
   RUNG wire#powerrail
      Contact( "SysDB_ZP_SeriesError_OP70".SeriesError[4].Error_present )
      S_Coil( "AnwDB_ZP_Alarm_OP70".FAULT[300] )
   END_RUNG
   // the same network as SCL:
   IF "SysDB_ZP_SeriesError_OP70".SeriesError[4].Error_present THEN
       "AnwDB_ZP_Alarm_OP70".FAULT[300] := TRUE;
   END_IF;
END_REGION

REGION Network 46: Alarm 301: Serial error 5 / Störmeldung 301: Serienfehler 5
   RUNG wire#powerrail
      Contact( "SysDB_ZP_SeriesError_OP70".SeriesError[5].Error_present )
      S_Coil( "AnwDB_ZP_Alarm_OP70".FAULT[301] )
   END_RUNG
   // the same network as SCL:
   IF "SysDB_ZP_SeriesError_OP70".SeriesError[5].Error_present THEN
       "AnwDB_ZP_Alarm_OP70".FAULT[301] := TRUE;
   END_IF;
END_REGION

REGION Network 47: Alarm 302: Serial error 6 / Störmeldung 302: Serienfehler 6
   RUNG wire#powerrail
      Contact( "SysDB_ZP_SeriesError_OP70".SeriesError[6].Error_present )
      S_Coil( "AnwDB_ZP_Alarm_OP70".FAULT[302] )
   END_RUNG
   // the same network as SCL:
   IF "SysDB_ZP_SeriesError_OP70".SeriesError[6].Error_present THEN
       "AnwDB_ZP_Alarm_OP70".FAULT[302] := TRUE;
   END_IF;
END_REGION

REGION Network 48: Alarm 303: Serial error 7 / Störmeldung 303: Serienfehler 7
   RUNG wire#powerrail
      Contact( "SysDB_ZP_SeriesError_OP70".SeriesError[7].Error_present )
      S_Coil( "AnwDB_ZP_Alarm_OP70".FAULT[303] )
   END_RUNG
   // the same network as SCL:
   IF "SysDB_ZP_SeriesError_OP70".SeriesError[7].Error_present THEN
       "AnwDB_ZP_Alarm_OP70".FAULT[303] := TRUE;
   END_IF;
END_REGION

REGION Network 49: Alarm 304: Serial error 8 / Störmeldung 304: Serienfehler 8
   RUNG wire#powerrail
      Contact( "SysDB_ZP_SeriesError_OP70".SeriesError[8].Error_present )
      S_Coil( "AnwDB_ZP_Alarm_OP70".FAULT[304] )
   END_RUNG
   // the same network as SCL:
   IF "SysDB_ZP_SeriesError_OP70".SeriesError[8].Error_present THEN
       "AnwDB_ZP_Alarm_OP70".FAULT[304] := TRUE;
   END_IF;
END_REGION

REGION Network 50: Alarm 305: Serial error 9 / Störmeldung 305: Serienfehler 9
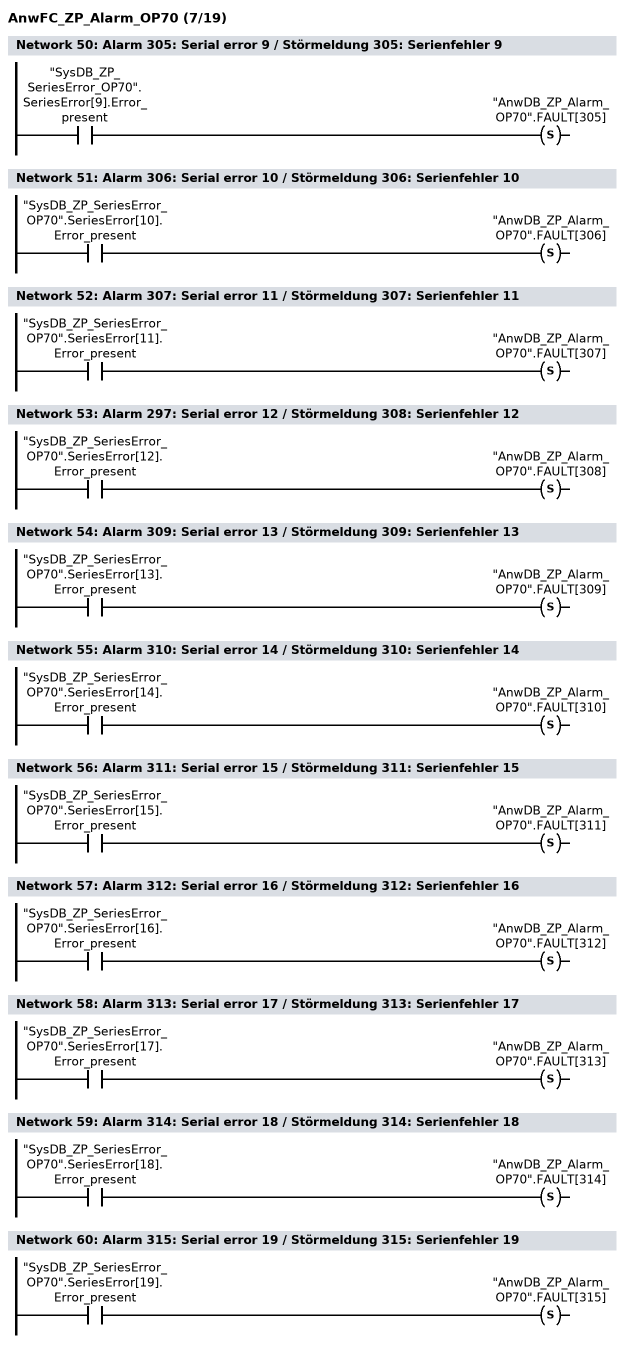
   RUNG wire#powerrail
      Contact( "SysDB_ZP_SeriesError_OP70".SeriesError[9].Error_present )
      S_Coil( "AnwDB_ZP_Alarm_OP70".FAULT[305] )
   END_RUNG
   // the same network as SCL:
   IF "SysDB_ZP_SeriesError_OP70".SeriesError[9].Error_present THEN
       "AnwDB_ZP_Alarm_OP70".FAULT[305] := TRUE;
   END_IF;
END_REGION

REGION Network 51: Alarm 306: Serial error 10 / Störmeldung 306: Serienfehler 10
   RUNG wire#powerrail
      Contact( "SysDB_ZP_SeriesError_OP70".SeriesError[10].Error_present )
      S_Coil( "AnwDB_ZP_Alarm_OP70".FAULT[306] )
   END_RUNG
   // the same network as SCL:
   IF "SysDB_ZP_SeriesError_OP70".SeriesError[10].Error_present THEN
       "AnwDB_ZP_Alarm_OP70".FAULT[306] := TRUE;
   END_IF;
END_REGION

REGION Network 52: Alarm 307: Serial error 11 / Störmeldung 307: Serienfehler 11
   RUNG wire#powerrail
      Contact( "SysDB_ZP_SeriesError_OP70".SeriesError[11].Error_present )
      S_Coil( "AnwDB_ZP_Alarm_OP70".FAULT[307] )
   END_RUNG
   // the same network as SCL:
   IF "SysDB_ZP_SeriesError_OP70".SeriesError[11].Error_present THEN
       "AnwDB_ZP_Alarm_OP70".FAULT[307] := TRUE;
   END_IF;
END_REGION

REGION Network 53: Alarm 297: Serial error 12 / Störmeldung 308: Serienfehler 12
   RUNG wire#powerrail
      Contact( "SysDB_ZP_SeriesError_OP70".SeriesError[12].Error_present )
      S_Coil( "AnwDB_ZP_Alarm_OP70".FAULT[308] )
   END_RUNG
   // the same network as SCL:
   IF "SysDB_ZP_SeriesError_OP70".SeriesError[12].Error_present THEN
       "AnwDB_ZP_Alarm_OP70".FAULT[308] := TRUE;
   END_IF;
END_REGION

REGION Network 54: Alarm 309: Serial error 13 / Störmeldung 309: Serienfehler 13
   RUNG wire#powerrail
      Contact( "SysDB_ZP_SeriesError_OP70".SeriesError[13].Error_present )
      S_Coil( "AnwDB_ZP_Alarm_OP70".FAULT[309] )
   END_RUNG
   // the same network as SCL:
   IF "SysDB_ZP_SeriesError_OP70".SeriesError[13].Error_present THEN
       "AnwDB_ZP_Alarm_OP70".FAULT[309] := TRUE;
   END_IF;
END_REGION

REGION Network 55: Alarm 310: Serial error 14 / Störmeldung 310: Serienfehler 14
   RUNG wire#powerrail
      Contact( "SysDB_ZP_SeriesError_OP70".SeriesError[14].Error_present )
      S_Coil( "AnwDB_ZP_Alarm_OP70".FAULT[310] )
   END_RUNG
   // the same network as SCL:
   IF "SysDB_ZP_SeriesError_OP70".SeriesError[14].Error_present THEN
       "AnwDB_ZP_Alarm_OP70".FAULT[310] := TRUE;
   END_IF;
END_REGION

REGION Network 56: Alarm 311: Serial error 15 / Störmeldung 311: Serienfehler 15
   RUNG wire#powerrail
      Contact( "SysDB_ZP_SeriesError_OP70".SeriesError[15].Error_present )
      S_Coil( "AnwDB_ZP_Alarm_OP70".FAULT[311] )
   END_RUNG
   // the same network as SCL:
   IF "SysDB_ZP_SeriesError_OP70".SeriesError[15].Error_present THEN
       "AnwDB_ZP_Alarm_OP70".FAULT[311] := TRUE;
   END_IF;
END_REGION

REGION Network 57: Alarm 312: Serial error 16 / Störmeldung 312: Serienfehler 16
   RUNG wire#powerrail
      Contact( "SysDB_ZP_SeriesError_OP70".SeriesError[16].Error_present )
      S_Coil( "AnwDB_ZP_Alarm_OP70".FAULT[312] )
   END_RUNG
   // the same network as SCL:
   IF "SysDB_ZP_SeriesError_OP70".SeriesError[16].Error_present THEN
       "AnwDB_ZP_Alarm_OP70".FAULT[312] := TRUE;
   END_IF;
END_REGION

REGION Network 58: Alarm 313: Serial error 17 / Störmeldung 313: Serienfehler 17
   RUNG wire#powerrail
      Contact( "SysDB_ZP_SeriesError_OP70".SeriesError[17].Error_present )
      S_Coil( "AnwDB_ZP_Alarm_OP70".FAULT[313] )
   END_RUNG
   // the same network as SCL:
   IF "SysDB_ZP_SeriesError_OP70".SeriesError[17].Error_present THEN
       "AnwDB_ZP_Alarm_OP70".FAULT[313] := TRUE;
   END_IF;
END_REGION

REGION Network 59: Alarm 314: Serial error 18 / Störmeldung 314: Serienfehler 18
   RUNG wire#powerrail
      Contact( "SysDB_ZP_SeriesError_OP70".SeriesError[18].Error_present )
      S_Coil( "AnwDB_ZP_Alarm_OP70".FAULT[314] )
   END_RUNG
   // the same network as SCL:
   IF "SysDB_ZP_SeriesError_OP70".SeriesError[18].Error_present THEN
       "AnwDB_ZP_Alarm_OP70".FAULT[314] := TRUE;
   END_IF;
END_REGION

REGION Network 60: Alarm 315: Serial error 19 / Störmeldung 315: Serienfehler 19
   RUNG wire#powerrail
      Contact( "SysDB_ZP_SeriesError_OP70".SeriesError[19].Error_present )
      S_Coil( "AnwDB_ZP_Alarm_OP70".FAULT[315] )
   END_RUNG
   // the same network as SCL:
   IF "SysDB_ZP_SeriesError_OP70".SeriesError[19].Error_present THEN
       "AnwDB_ZP_Alarm_OP70".FAULT[315] := TRUE;
   END_IF;
END_REGION

REGION Network 61: Alarm 316: Serial error 20 / Störmeldung 316: Serienfehler 20
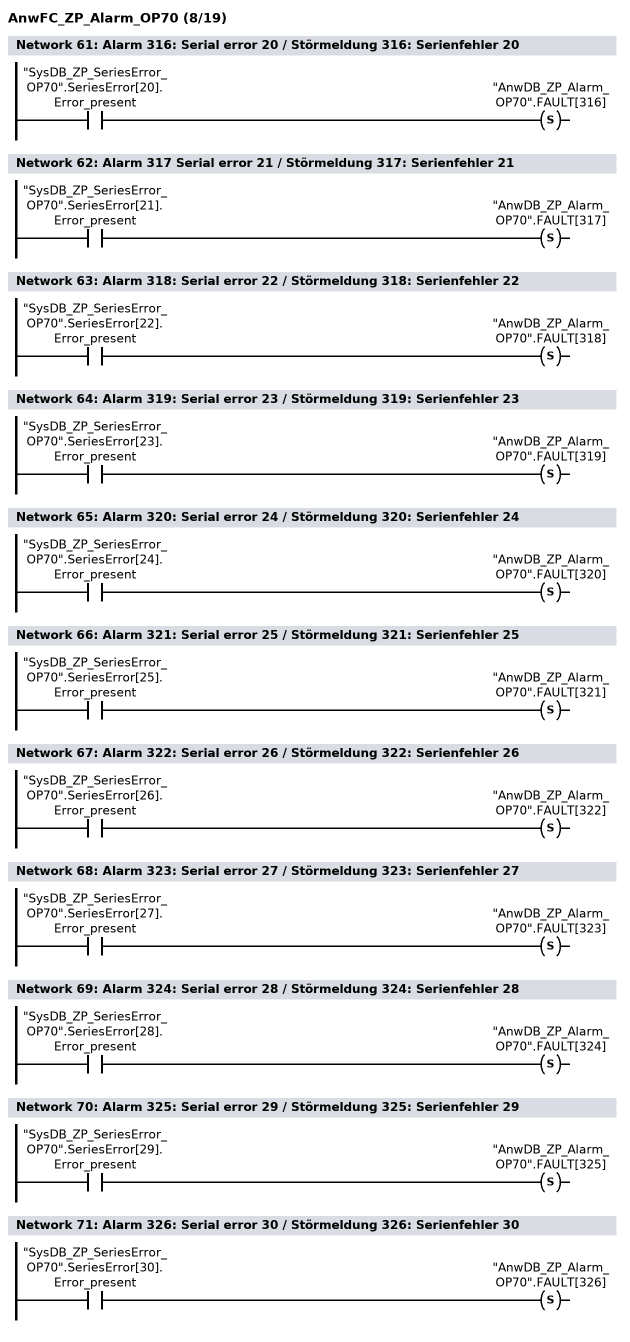
   RUNG wire#powerrail
      Contact( "SysDB_ZP_SeriesError_OP70".SeriesError[20].Error_present )
      S_Coil( "AnwDB_ZP_Alarm_OP70".FAULT[316] )
   END_RUNG
   // the same network as SCL:
   IF "SysDB_ZP_SeriesError_OP70".SeriesError[20].Error_present THEN
       "AnwDB_ZP_Alarm_OP70".FAULT[316] := TRUE;
   END_IF;
END_REGION

REGION Network 62: Alarm 317 Serial error 21 / Störmeldung 317: Serienfehler 21
   RUNG wire#powerrail
      Contact( "SysDB_ZP_SeriesError_OP70".SeriesError[21].Error_present )
      S_Coil( "AnwDB_ZP_Alarm_OP70".FAULT[317] )
   END_RUNG
   // the same network as SCL:
   IF "SysDB_ZP_SeriesError_OP70".SeriesError[21].Error_present THEN
       "AnwDB_ZP_Alarm_OP70".FAULT[317] := TRUE;
   END_IF;
END_REGION

REGION Network 63: Alarm 318: Serial error 22 / Störmeldung 318: Serienfehler 22
   RUNG wire#powerrail
      Contact( "SysDB_ZP_SeriesError_OP70".SeriesError[22].Error_present )
      S_Coil( "AnwDB_ZP_Alarm_OP70".FAULT[318] )
   END_RUNG
   // the same network as SCL:
   IF "SysDB_ZP_SeriesError_OP70".SeriesError[22].Error_present THEN
       "AnwDB_ZP_Alarm_OP70".FAULT[318] := TRUE;
   END_IF;
END_REGION

REGION Network 64: Alarm 319: Serial error 23 / Störmeldung 319: Serienfehler 23
   RUNG wire#powerrail
      Contact( "SysDB_ZP_SeriesError_OP70".SeriesError[23].Error_present )
      S_Coil( "AnwDB_ZP_Alarm_OP70".FAULT[319] )
   END_RUNG
   // the same network as SCL:
   IF "SysDB_ZP_SeriesError_OP70".SeriesError[23].Error_present THEN
       "AnwDB_ZP_Alarm_OP70".FAULT[319] := TRUE;
   END_IF;
END_REGION

REGION Network 65: Alarm 320: Serial error 24 / Störmeldung 320: Serienfehler 24
   RUNG wire#powerrail
      Contact( "SysDB_ZP_SeriesError_OP70".SeriesError[24].Error_present )
      S_Coil( "AnwDB_ZP_Alarm_OP70".FAULT[320] )
   END_RUNG
   // the same network as SCL:
   IF "SysDB_ZP_SeriesError_OP70".SeriesError[24].Error_present THEN
       "AnwDB_ZP_Alarm_OP70".FAULT[320] := TRUE;
   END_IF;
END_REGION

REGION Network 66: Alarm 321: Serial error 25 / Störmeldung 321: Serienfehler 25
   RUNG wire#powerrail
      Contact( "SysDB_ZP_SeriesError_OP70".SeriesError[25].Error_present )
      S_Coil( "AnwDB_ZP_Alarm_OP70".FAULT[321] )
   END_RUNG
   // the same network as SCL:
   IF "SysDB_ZP_SeriesError_OP70".SeriesError[25].Error_present THEN
       "AnwDB_ZP_Alarm_OP70".FAULT[321] := TRUE;
   END_IF;
END_REGION

REGION Network 67: Alarm 322: Serial error 26 / Störmeldung 322: Serienfehler 26
   RUNG wire#powerrail
      Contact( "SysDB_ZP_SeriesError_OP70".SeriesError[26].Error_present )
      S_Coil( "AnwDB_ZP_Alarm_OP70".FAULT[322] )
   END_RUNG
   // the same network as SCL:
   IF "SysDB_ZP_SeriesError_OP70".SeriesError[26].Error_present THEN
       "AnwDB_ZP_Alarm_OP70".FAULT[322] := TRUE;
   END_IF;
END_REGION

REGION Network 68: Alarm 323: Serial error 27 / Störmeldung 323: Serienfehler 27
   RUNG wire#powerrail
      Contact( "SysDB_ZP_SeriesError_OP70".SeriesError[27].Error_present )
      S_Coil( "AnwDB_ZP_Alarm_OP70".FAULT[323] )
   END_RUNG
   // the same network as SCL:
   IF "SysDB_ZP_SeriesError_OP70".SeriesError[27].Error_present THEN
       "AnwDB_ZP_Alarm_OP70".FAULT[323] := TRUE;
   END_IF;
END_REGION

REGION Network 69: Alarm 324: Serial error 28 / Störmeldung 324: Serienfehler 28
   RUNG wire#powerrail
      Contact( "SysDB_ZP_SeriesError_OP70".SeriesError[28].Error_present )
      S_Coil( "AnwDB_ZP_Alarm_OP70".FAULT[324] )
   END_RUNG
   // the same network as SCL:
   IF "SysDB_ZP_SeriesError_OP70".SeriesError[28].Error_present THEN
       "AnwDB_ZP_Alarm_OP70".FAULT[324] := TRUE;
   END_IF;
END_REGION

REGION Network 70: Alarm 325: Serial error 29 / Störmeldung 325: Serienfehler 29
   RUNG wire#powerrail
      Contact( "SysDB_ZP_SeriesError_OP70".SeriesError[29].Error_present )
      S_Coil( "AnwDB_ZP_Alarm_OP70".FAULT[325] )
   END_RUNG
   // the same network as SCL:
   IF "SysDB_ZP_SeriesError_OP70".SeriesError[29].Error_present THEN
       "AnwDB_ZP_Alarm_OP70".FAULT[325] := TRUE;
   END_IF;
END_REGION

REGION Network 71: Alarm 326: Serial error 30 / Störmeldung 326: Serienfehler 30
   RUNG wire#powerrail
      Contact( "SysDB_ZP_SeriesError_OP70".SeriesError[30].Error_present )
      S_Coil( "AnwDB_ZP_Alarm_OP70".FAULT[326] )
   END_RUNG
   // the same network as SCL:
   IF "SysDB_ZP_SeriesError_OP70".SeriesError[30].Error_present THEN
       "AnwDB_ZP_Alarm_OP70".FAULT[326] := TRUE;
   END_IF;
END_REGION

REGION Network 72: Alarm 327: Serial error 31 / Störmeldung 327: Serienfehler 31
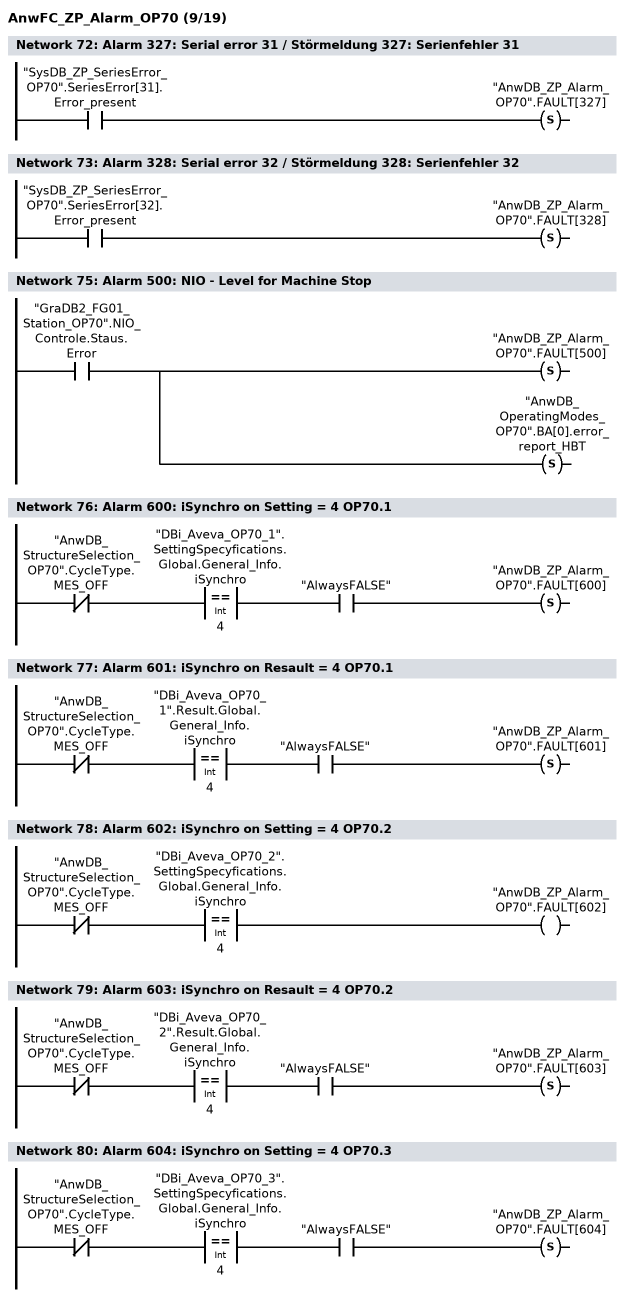
   RUNG wire#powerrail
      Contact( "SysDB_ZP_SeriesError_OP70".SeriesError[31].Error_present )
      S_Coil( "AnwDB_ZP_Alarm_OP70".FAULT[327] )
   END_RUNG
   // the same network as SCL:
   IF "SysDB_ZP_SeriesError_OP70".SeriesError[31].Error_present THEN
       "AnwDB_ZP_Alarm_OP70".FAULT[327] := TRUE;
   END_IF;
END_REGION

REGION Network 73: Alarm 328: Serial error 32 / Störmeldung 328: Serienfehler 32
   RUNG wire#powerrail
      Contact( "SysDB_ZP_SeriesError_OP70".SeriesError[32].Error_present )
      S_Coil( "AnwDB_ZP_Alarm_OP70".FAULT[328] )
   END_RUNG
   // the same network as SCL:
   IF "SysDB_ZP_SeriesError_OP70".SeriesError[32].Error_present THEN
       "AnwDB_ZP_Alarm_OP70".FAULT[328] := TRUE;
   END_IF;
END_REGION

REGION Network 74: Alarm 341 - 424 Reserved for pair fault / Störmeldung 341 - 424: Reserviert für Paarfehler
   // Alarm 341 - 424 Reserved for pair fault / Störung 341 -  424 Reserviert für Paarfehler
END_REGION

REGION Network 75: Alarm 500: NIO - Level for Machine Stop
   RUNG wire#powerrail
      Contact( "GraDB2_FG01_Station_OP70".NIO_Controle.Staus.Error )
      wire#w1
      S_Coil( "AnwDB_ZP_Alarm_OP70".FAULT[500] )
   END_RUNG
   RUNG wire#w1
      S_Coil( "AnwDB_OperatingModes_OP70".BA[0].error_report_HBT )
   END_RUNG
   // the same network as SCL:
   IF "GraDB2_FG01_Station_OP70".NIO_Controle.Staus.Error THEN
       "AnwDB_ZP_Alarm_OP70".FAULT[500] := TRUE;
       "AnwDB_OperatingModes_OP70".BA[0].error_report_HBT := TRUE;
   END_IF;
END_REGION

REGION Network 76: Alarm 600: iSynchro on Setting = 4 OP70.1
   RUNG wire#powerrail
      I_Contact( "AnwDB_StructureSelection_OP70".CycleType.MES_OFF )
      { S7_Templates := "SrcType := Int" } EQ_Contact(in1 := "DBi_Aveva_OP70_1".SettingSpecyfications.Global.General_Info.iSynchro, in2 := 4)
      Contact( "AlwaysFALSE" )
      S_Coil( "AnwDB_ZP_Alarm_OP70".FAULT[600] )
   END_RUNG
   // the same network as SCL:
   IF NOT "AnwDB_StructureSelection_OP70".CycleType.MES_OFF AND ("DBi_Aveva_OP70_1".SettingSpecyfications.Global.General_Info.iSynchro = 4) AND "AlwaysFALSE" THEN
       "AnwDB_ZP_Alarm_OP70".FAULT[600] := TRUE;
   END_IF;
END_REGION

REGION Network 77: Alarm 601: iSynchro on Resault = 4 OP70.1
   RUNG wire#powerrail
      I_Contact( "AnwDB_StructureSelection_OP70".CycleType.MES_OFF )
      { S7_Templates := "SrcType := Int" } EQ_Contact(in1 := "DBi_Aveva_OP70_1".Result.Global.General_Info.iSynchro, in2 := 4)
      Contact( "AlwaysFALSE" )
      S_Coil( "AnwDB_ZP_Alarm_OP70".FAULT[601] )
   END_RUNG
   // the same network as SCL:
   IF NOT "AnwDB_StructureSelection_OP70".CycleType.MES_OFF AND ("DBi_Aveva_OP70_1".Result.Global.General_Info.iSynchro = 4) AND "AlwaysFALSE" THEN
       "AnwDB_ZP_Alarm_OP70".FAULT[601] := TRUE;
   END_IF;
END_REGION

REGION Network 78: Alarm 602: iSynchro on Setting = 4 OP70.2
   RUNG wire#powerrail
      I_Contact( "AnwDB_StructureSelection_OP70".CycleType.MES_OFF )
      { S7_Templates := "SrcType := Int" } EQ_Contact(in1 := "DBi_Aveva_OP70_2".SettingSpecyfications.Global.General_Info.iSynchro, in2 := 4)
      Coil( "AnwDB_ZP_Alarm_OP70".FAULT[602] )
   END_RUNG
   // the same network as SCL:
   "AnwDB_ZP_Alarm_OP70".FAULT[602] := NOT "AnwDB_StructureSelection_OP70".CycleType.MES_OFF AND ("DBi_Aveva_OP70_2".SettingSpecyfications.Global.General_Info.iSynchro = 4);
END_REGION

REGION Network 79: Alarm 603: iSynchro on Resault = 4 OP70.2
   RUNG wire#powerrail
      I_Contact( "AnwDB_StructureSelection_OP70".CycleType.MES_OFF )
      { S7_Templates := "SrcType := Int" } EQ_Contact(in1 := "DBi_Aveva_OP70_2".Result.Global.General_Info.iSynchro, in2 := 4)
      Contact( "AlwaysFALSE" )
      S_Coil( "AnwDB_ZP_Alarm_OP70".FAULT[603] )
   END_RUNG
   // the same network as SCL:
   IF NOT "AnwDB_StructureSelection_OP70".CycleType.MES_OFF AND ("DBi_Aveva_OP70_2".Result.Global.General_Info.iSynchro = 4) AND "AlwaysFALSE" THEN
       "AnwDB_ZP_Alarm_OP70".FAULT[603] := TRUE;
   END_IF;
END_REGION

REGION Network 80: Alarm 604: iSynchro on Setting = 4 OP70.3
   RUNG wire#powerrail
      I_Contact( "AnwDB_StructureSelection_OP70".CycleType.MES_OFF )
      { S7_Templates := "SrcType := Int" } EQ_Contact(in1 := "DBi_Aveva_OP70_3".SettingSpecyfications.Global.General_Info.iSynchro, in2 := 4)
      Contact( "AlwaysFALSE" )
      S_Coil( "AnwDB_ZP_Alarm_OP70".FAULT[604] )
   END_RUNG
   // the same network as SCL:
   IF NOT "AnwDB_StructureSelection_OP70".CycleType.MES_OFF AND ("DBi_Aveva_OP70_3".SettingSpecyfications.Global.General_Info.iSynchro = 4) AND "AlwaysFALSE" THEN
       "AnwDB_ZP_Alarm_OP70".FAULT[604] := TRUE;
   END_IF;
END_REGION

REGION Network 81: Alarm 605: iSynchro on Resault = 4 OP70.3
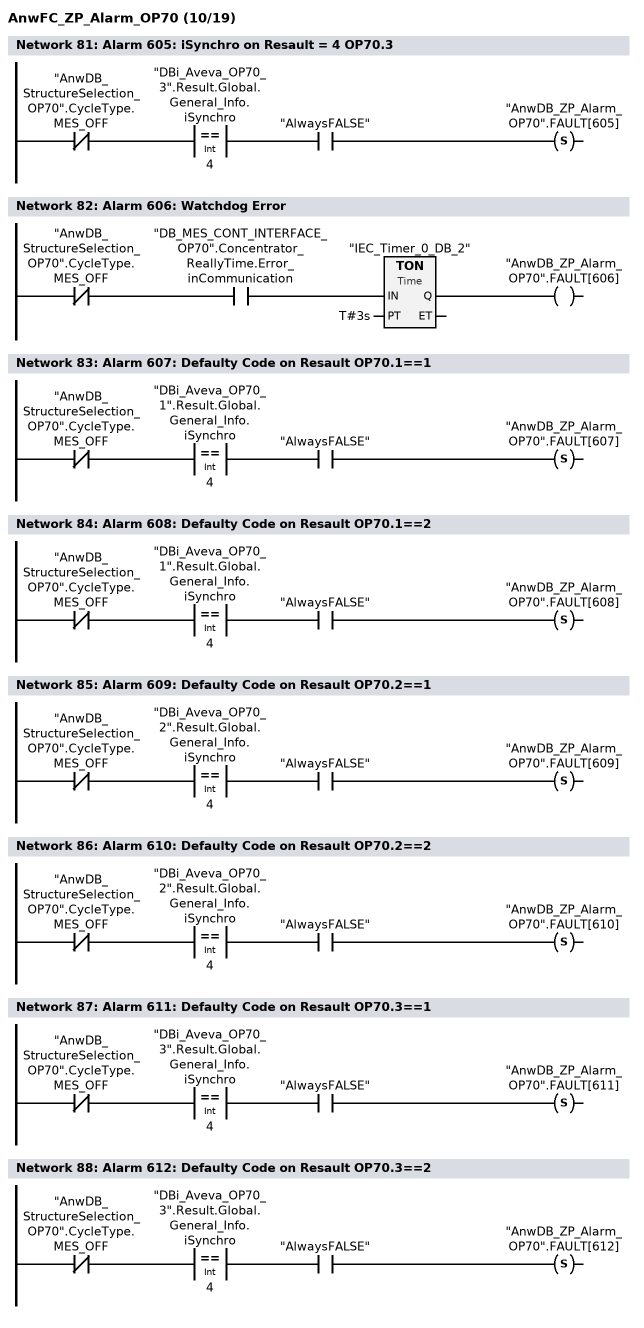
   RUNG wire#powerrail
      I_Contact( "AnwDB_StructureSelection_OP70".CycleType.MES_OFF )
      { S7_Templates := "SrcType := Int" } EQ_Contact(in1 := "DBi_Aveva_OP70_3".Result.Global.General_Info.iSynchro, in2 := 4)
      Contact( "AlwaysFALSE" )
      S_Coil( "AnwDB_ZP_Alarm_OP70".FAULT[605] )
   END_RUNG
   // the same network as SCL:
   IF NOT "AnwDB_StructureSelection_OP70".CycleType.MES_OFF AND ("DBi_Aveva_OP70_3".Result.Global.General_Info.iSynchro = 4) AND "AlwaysFALSE" THEN
       "AnwDB_ZP_Alarm_OP70".FAULT[605] := TRUE;
   END_IF;
END_REGION

REGION Network 82: Alarm 606: Watchdog Error
   RUNG wire#powerrail
      I_Contact( "AnwDB_StructureSelection_OP70".CycleType.MES_OFF )
      Contact( "DB_MES_CONT_INTERFACE_OP70".Concentrator_ReallyTime.Error_inCommunication )
      { S7_Templates := "time_type := Time" } "IEC_Timer_0_DB_2".TON(pt := T#3s, et =>)
      Coil( "AnwDB_ZP_Alarm_OP70".FAULT[606] )
   END_RUNG
   // the same network as SCL:
   "IEC_Timer_0_DB_2".TON(IN := NOT "AnwDB_StructureSelection_OP70".CycleType.MES_OFF AND "DB_MES_CONT_INTERFACE_OP70".Concentrator_ReallyTime.Error_inCommunication,
                          PT := T#3s);
   "AnwDB_ZP_Alarm_OP70".FAULT[606] := "IEC_Timer_0_DB_2".Q;
END_REGION

REGION Network 83: Alarm 607: Defaulty Code on Resault OP70.1==1
   RUNG wire#powerrail
      I_Contact( "AnwDB_StructureSelection_OP70".CycleType.MES_OFF )
      { S7_Templates := "SrcType := Int" } EQ_Contact(in1 := "DBi_Aveva_OP70_1".Result.Global.General_Info.iSynchro, in2 := 4)
      Contact( "AlwaysFALSE" )
      S_Coil( "AnwDB_ZP_Alarm_OP70".FAULT[607] )
   END_RUNG
   // the same network as SCL:
   IF NOT "AnwDB_StructureSelection_OP70".CycleType.MES_OFF AND ("DBi_Aveva_OP70_1".Result.Global.General_Info.iSynchro = 4) AND "AlwaysFALSE" THEN
       "AnwDB_ZP_Alarm_OP70".FAULT[607] := TRUE;
   END_IF;
END_REGION

REGION Network 84: Alarm 608: Defaulty Code on Resault OP70.1==2
   RUNG wire#powerrail
      I_Contact( "AnwDB_StructureSelection_OP70".CycleType.MES_OFF )
      { S7_Templates := "SrcType := Int" } EQ_Contact(in1 := "DBi_Aveva_OP70_1".Result.Global.General_Info.iSynchro, in2 := 4)
      Contact( "AlwaysFALSE" )
      S_Coil( "AnwDB_ZP_Alarm_OP70".FAULT[608] )
   END_RUNG
   // the same network as SCL:
   IF NOT "AnwDB_StructureSelection_OP70".CycleType.MES_OFF AND ("DBi_Aveva_OP70_1".Result.Global.General_Info.iSynchro = 4) AND "AlwaysFALSE" THEN
       "AnwDB_ZP_Alarm_OP70".FAULT[608] := TRUE;
   END_IF;
END_REGION

REGION Network 85: Alarm 609: Defaulty Code on Resault OP70.2==1
   RUNG wire#powerrail
      I_Contact( "AnwDB_StructureSelection_OP70".CycleType.MES_OFF )
      { S7_Templates := "SrcType := Int" } EQ_Contact(in1 := "DBi_Aveva_OP70_2".Result.Global.General_Info.iSynchro, in2 := 4)
      Contact( "AlwaysFALSE" )
      S_Coil( "AnwDB_ZP_Alarm_OP70".FAULT[609] )
   END_RUNG
   // the same network as SCL:
   IF NOT "AnwDB_StructureSelection_OP70".CycleType.MES_OFF AND ("DBi_Aveva_OP70_2".Result.Global.General_Info.iSynchro = 4) AND "AlwaysFALSE" THEN
       "AnwDB_ZP_Alarm_OP70".FAULT[609] := TRUE;
   END_IF;
END_REGION

REGION Network 86: Alarm 610: Defaulty Code on Resault OP70.2==2
   RUNG wire#powerrail
      I_Contact( "AnwDB_StructureSelection_OP70".CycleType.MES_OFF )
      { S7_Templates := "SrcType := Int" } EQ_Contact(in1 := "DBi_Aveva_OP70_2".Result.Global.General_Info.iSynchro, in2 := 4)
      Contact( "AlwaysFALSE" )
      S_Coil( "AnwDB_ZP_Alarm_OP70".FAULT[610] )
   END_RUNG
   // the same network as SCL:
   IF NOT "AnwDB_StructureSelection_OP70".CycleType.MES_OFF AND ("DBi_Aveva_OP70_2".Result.Global.General_Info.iSynchro = 4) AND "AlwaysFALSE" THEN
       "AnwDB_ZP_Alarm_OP70".FAULT[610] := TRUE;
   END_IF;
END_REGION

REGION Network 87: Alarm 611: Defaulty Code on Resault OP70.3==1
   RUNG wire#powerrail
      I_Contact( "AnwDB_StructureSelection_OP70".CycleType.MES_OFF )
      { S7_Templates := "SrcType := Int" } EQ_Contact(in1 := "DBi_Aveva_OP70_3".Result.Global.General_Info.iSynchro, in2 := 4)
      Contact( "AlwaysFALSE" )
      S_Coil( "AnwDB_ZP_Alarm_OP70".FAULT[611] )
   END_RUNG
   // the same network as SCL:
   IF NOT "AnwDB_StructureSelection_OP70".CycleType.MES_OFF AND ("DBi_Aveva_OP70_3".Result.Global.General_Info.iSynchro = 4) AND "AlwaysFALSE" THEN
       "AnwDB_ZP_Alarm_OP70".FAULT[611] := TRUE;
   END_IF;
END_REGION

REGION Network 88: Alarm 612: Defaulty Code on Resault OP70.3==2
   RUNG wire#powerrail
      I_Contact( "AnwDB_StructureSelection_OP70".CycleType.MES_OFF )
      { S7_Templates := "SrcType := Int" } EQ_Contact(in1 := "DBi_Aveva_OP70_3".Result.Global.General_Info.iSynchro, in2 := 4)
      Contact( "AlwaysFALSE" )
      S_Coil( "AnwDB_ZP_Alarm_OP70".FAULT[612] )
   END_RUNG
   // the same network as SCL:
   IF NOT "AnwDB_StructureSelection_OP70".CycleType.MES_OFF AND ("DBi_Aveva_OP70_3".Result.Global.General_Info.iSynchro = 4) AND "AlwaysFALSE" THEN
       "AnwDB_ZP_Alarm_OP70".FAULT[612] := TRUE;
   END_IF;
END_REGION

REGION Network 89: Alarm 613: Defaulty Code on Setting OP70.1==1
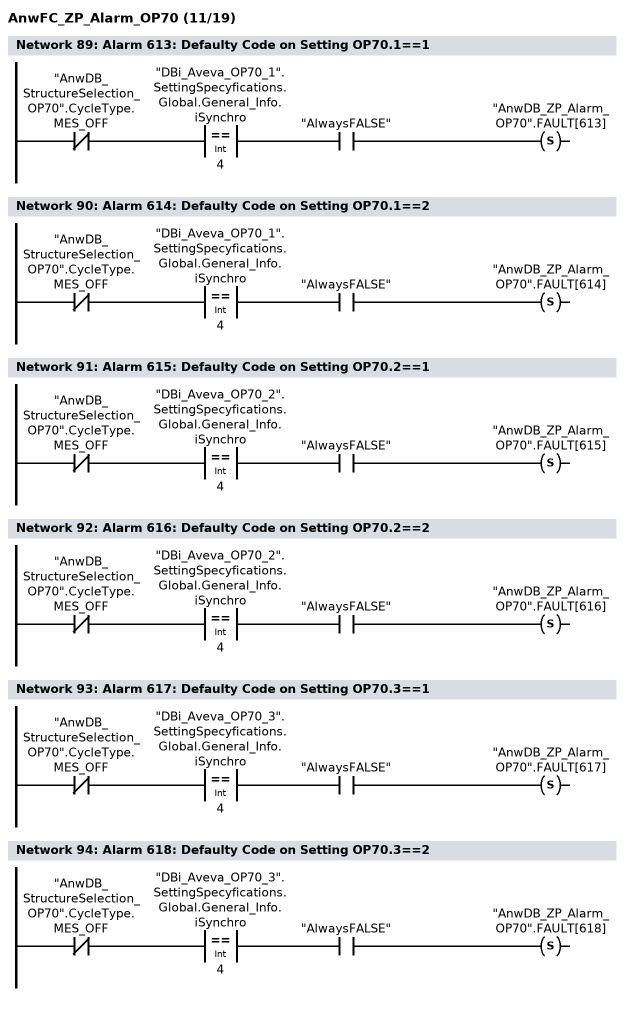
   RUNG wire#powerrail
      I_Contact( "AnwDB_StructureSelection_OP70".CycleType.MES_OFF )
      { S7_Templates := "SrcType := Int" } EQ_Contact(in1 := "DBi_Aveva_OP70_1".SettingSpecyfications.Global.General_Info.iSynchro, in2 := 4)
      Contact( "AlwaysFALSE" )
      S_Coil( "AnwDB_ZP_Alarm_OP70".FAULT[613] )
   END_RUNG
   // the same network as SCL:
   IF NOT "AnwDB_StructureSelection_OP70".CycleType.MES_OFF AND ("DBi_Aveva_OP70_1".SettingSpecyfications.Global.General_Info.iSynchro = 4) AND "AlwaysFALSE" THEN
       "AnwDB_ZP_Alarm_OP70".FAULT[613] := TRUE;
   END_IF;
END_REGION

REGION Network 90: Alarm 614: Defaulty Code on Setting OP70.1==2
   RUNG wire#powerrail
      I_Contact( "AnwDB_StructureSelection_OP70".CycleType.MES_OFF )
      { S7_Templates := "SrcType := Int" } EQ_Contact(in1 := "DBi_Aveva_OP70_1".SettingSpecyfications.Global.General_Info.iSynchro, in2 := 4)
      Contact( "AlwaysFALSE" )
      S_Coil( "AnwDB_ZP_Alarm_OP70".FAULT[614] )
   END_RUNG
   // the same network as SCL:
   IF NOT "AnwDB_StructureSelection_OP70".CycleType.MES_OFF AND ("DBi_Aveva_OP70_1".SettingSpecyfications.Global.General_Info.iSynchro = 4) AND "AlwaysFALSE" THEN
       "AnwDB_ZP_Alarm_OP70".FAULT[614] := TRUE;
   END_IF;
END_REGION

REGION Network 91: Alarm 615: Defaulty Code on Setting OP70.2==1
   RUNG wire#powerrail
      I_Contact( "AnwDB_StructureSelection_OP70".CycleType.MES_OFF )
      { S7_Templates := "SrcType := Int" } EQ_Contact(in1 := "DBi_Aveva_OP70_2".SettingSpecyfications.Global.General_Info.iSynchro, in2 := 4)
      Contact( "AlwaysFALSE" )
      S_Coil( "AnwDB_ZP_Alarm_OP70".FAULT[615] )
   END_RUNG
   // the same network as SCL:
   IF NOT "AnwDB_StructureSelection_OP70".CycleType.MES_OFF AND ("DBi_Aveva_OP70_2".SettingSpecyfications.Global.General_Info.iSynchro = 4) AND "AlwaysFALSE" THEN
       "AnwDB_ZP_Alarm_OP70".FAULT[615] := TRUE;
   END_IF;
END_REGION

REGION Network 92: Alarm 616: Defaulty Code on Setting OP70.2==2
   RUNG wire#powerrail
      I_Contact( "AnwDB_StructureSelection_OP70".CycleType.MES_OFF )
      { S7_Templates := "SrcType := Int" } EQ_Contact(in1 := "DBi_Aveva_OP70_2".SettingSpecyfications.Global.General_Info.iSynchro, in2 := 4)
      Contact( "AlwaysFALSE" )
      S_Coil( "AnwDB_ZP_Alarm_OP70".FAULT[616] )
   END_RUNG
   // the same network as SCL:
   IF NOT "AnwDB_StructureSelection_OP70".CycleType.MES_OFF AND ("DBi_Aveva_OP70_2".SettingSpecyfications.Global.General_Info.iSynchro = 4) AND "AlwaysFALSE" THEN
       "AnwDB_ZP_Alarm_OP70".FAULT[616] := TRUE;
   END_IF;
END_REGION

REGION Network 93: Alarm 617: Defaulty Code on Setting OP70.3==1
   RUNG wire#powerrail
      I_Contact( "AnwDB_StructureSelection_OP70".CycleType.MES_OFF )
      { S7_Templates := "SrcType := Int" } EQ_Contact(in1 := "DBi_Aveva_OP70_3".SettingSpecyfications.Global.General_Info.iSynchro, in2 := 4)
      Contact( "AlwaysFALSE" )
      S_Coil( "AnwDB_ZP_Alarm_OP70".FAULT[617] )
   END_RUNG
   // the same network as SCL:
   IF NOT "AnwDB_StructureSelection_OP70".CycleType.MES_OFF AND ("DBi_Aveva_OP70_3".SettingSpecyfications.Global.General_Info.iSynchro = 4) AND "AlwaysFALSE" THEN
       "AnwDB_ZP_Alarm_OP70".FAULT[617] := TRUE;
   END_IF;
END_REGION

REGION Network 94: Alarm 618: Defaulty Code on Setting OP70.3==2
   RUNG wire#powerrail
      I_Contact( "AnwDB_StructureSelection_OP70".CycleType.MES_OFF )
      { S7_Templates := "SrcType := Int" } EQ_Contact(in1 := "DBi_Aveva_OP70_3".SettingSpecyfications.Global.General_Info.iSynchro, in2 := 4)
      Contact( "AlwaysFALSE" )
      S_Coil( "AnwDB_ZP_Alarm_OP70".FAULT[618] )
   END_RUNG
   // the same network as SCL:
   IF NOT "AnwDB_StructureSelection_OP70".CycleType.MES_OFF AND ("DBi_Aveva_OP70_3".SettingSpecyfications.Global.General_Info.iSynchro = 4) AND "AlwaysFALSE" THEN
       "AnwDB_ZP_Alarm_OP70".FAULT[618] := TRUE;
   END_IF;
END_REGION

REGION Network 95: Alarm 800: Camera - Component not detected
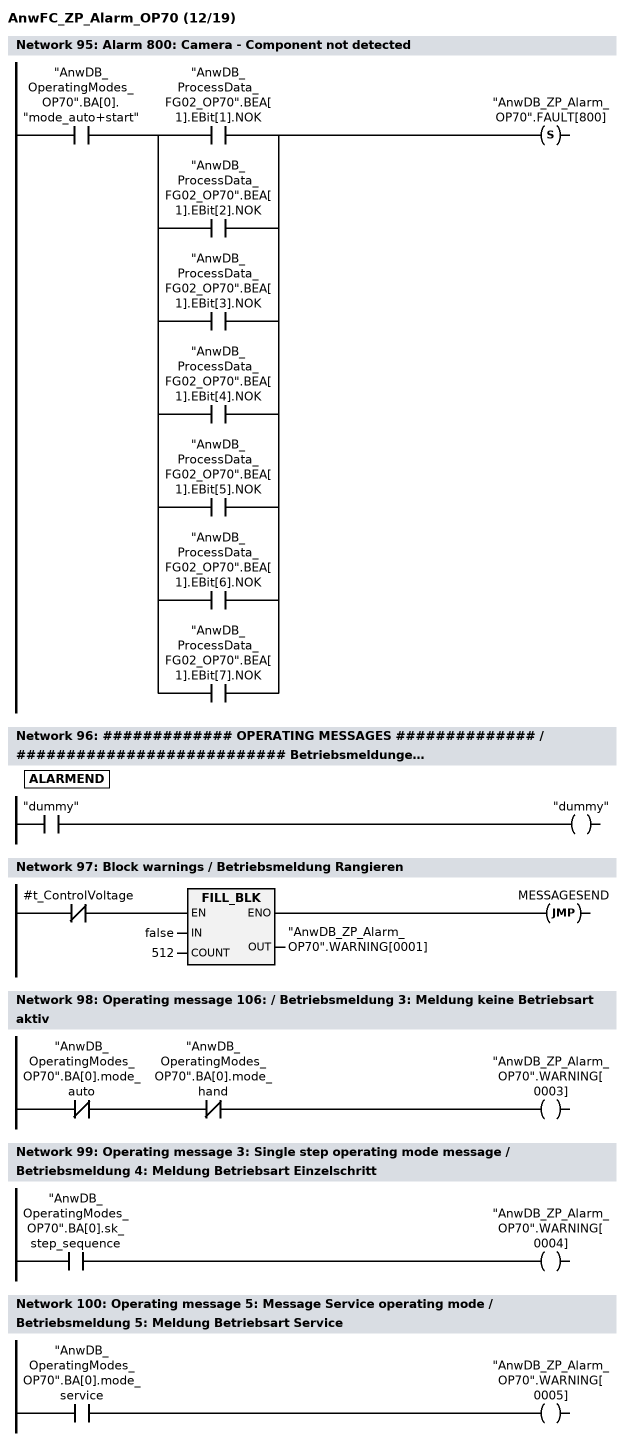
   RUNG wire#powerrail
      Contact( "AnwDB_OperatingModes_OP70".BA[0]."mode_auto+start" )
      wire#w1
      Contact( "AnwDB_ProcessData_FG02_OP70".BEA[1].EBit[1].NOK )
      wire#w2
      S_Coil( "AnwDB_ZP_Alarm_OP70".FAULT[800] )
   END_RUNG
   RUNG wire#w1
      Contact( "AnwDB_ProcessData_FG02_OP70".BEA[1].EBit[2].NOK )
   END_RUNG wire#w2
   RUNG wire#w1
      Contact( "AnwDB_ProcessData_FG02_OP70".BEA[1].EBit[3].NOK )
   END_RUNG wire#w2
   RUNG wire#w1
      Contact( "AnwDB_ProcessData_FG02_OP70".BEA[1].EBit[4].NOK )
   END_RUNG wire#w2
   RUNG wire#w1
      Contact( "AnwDB_ProcessData_FG02_OP70".BEA[1].EBit[5].NOK )
   END_RUNG wire#w2
   RUNG wire#w1
      Contact( "AnwDB_ProcessData_FG02_OP70".BEA[1].EBit[6].NOK )
   END_RUNG wire#w2
   RUNG wire#w1
      Contact( "AnwDB_ProcessData_FG02_OP70".BEA[1].EBit[7].NOK )
   END_RUNG wire#w2
   // the same network as SCL:
   IF "AnwDB_OperatingModes_OP70".BA[0]."mode_auto+start" AND ("AnwDB_ProcessData_FG02_OP70".BEA[1].EBit[1].NOK OR "AnwDB_ProcessData_FG02_OP70".BEA[1].EBit[2].NOK OR "AnwDB_ProcessData_FG02_OP70".BEA[1].EBit[3].NOK OR "AnwDB_ProcessData_FG02_OP70".BEA[1].EBit[4].NOK OR "AnwDB_ProcessData_FG02_OP70".BEA[1].EBit[5].NOK OR "AnwDB_ProcessData_FG02_OP70".BEA[1].EBit[6].NOK OR "AnwDB_ProcessData_FG02_OP70".BEA[1].EBit[7].NOK) THEN
       "AnwDB_ZP_Alarm_OP70".FAULT[800] := TRUE;
   END_IF;
END_REGION

REGION Network 96: ############# OPERATING MESSAGES ############## / ########################### Betriebsmeldungen ##########################
   Label( ALARMEND )
   RUNG wire#powerrail
      Contact( "dummy" )
      Coil( "dummy" )
   END_RUNG
   // the same network as SCL:
   ALARMEND:
   "dummy" := "dummy";
END_REGION

REGION Network 97: Block warnings / Betriebsmeldung Rangieren
   RUNG wire#powerrail
      I_Contact( #t_ControlVoltage )
      FillBlockI(in := false, count := 512, out => "AnwDB_ZP_Alarm_OP70".WARNING[0001])
      JumpCoil( MESSAGESEND )
   END_RUNG
   // the same network as SCL:
   IF NOT #t_ControlVoltage THEN
       FILL_BLK(IN := false, COUNT := 512, OUT => "AnwDB_ZP_Alarm_OP70".WARNING[0001]);
       GOTO MESSAGESEND;
   END_IF;
END_REGION

REGION Network 98: Operating message 106: / Betriebsmeldung 3: Meldung keine Betriebsart aktiv
   RUNG wire#powerrail
      I_Contact( "AnwDB_OperatingModes_OP70".BA[0].mode_auto )
      I_Contact( "AnwDB_OperatingModes_OP70".BA[0].mode_hand )
      Coil( "AnwDB_ZP_Alarm_OP70".WARNING[0003] )
   END_RUNG
   // the same network as SCL:
   "AnwDB_ZP_Alarm_OP70".WARNING[0003] := NOT "AnwDB_OperatingModes_OP70".BA[0].mode_auto AND NOT "AnwDB_OperatingModes_OP70".BA[0].mode_hand;
END_REGION

REGION Network 99: Operating message 3: Single step operating mode message / Betriebsmeldung 4: Meldung Betriebsart Einzelschritt
   RUNG wire#powerrail
      Contact( "AnwDB_OperatingModes_OP70".BA[0].sk_step_sequence )
      Coil( "AnwDB_ZP_Alarm_OP70".WARNING[0004] )
   END_RUNG
   // the same network as SCL:
   "AnwDB_ZP_Alarm_OP70".WARNING[0004] := "AnwDB_OperatingModes_OP70".BA[0].sk_step_sequence;
END_REGION

REGION Network 100: Operating message 5: Message Service operating mode / Betriebsmeldung 5: Meldung Betriebsart Service
   RUNG wire#powerrail
      Contact( "AnwDB_OperatingModes_OP70".BA[0].mode_service )
      Coil( "AnwDB_ZP_Alarm_OP70".WARNING[0005] )
   END_RUNG
   // the same network as SCL:
   "AnwDB_ZP_Alarm_OP70".WARNING[0005] := "AnwDB_OperatingModes_OP70".BA[0].mode_service;
END_REGION

REGION Network 101: Operating message 6: Message Type change / Betriebsmeldung 6: Typwechsel aktiv
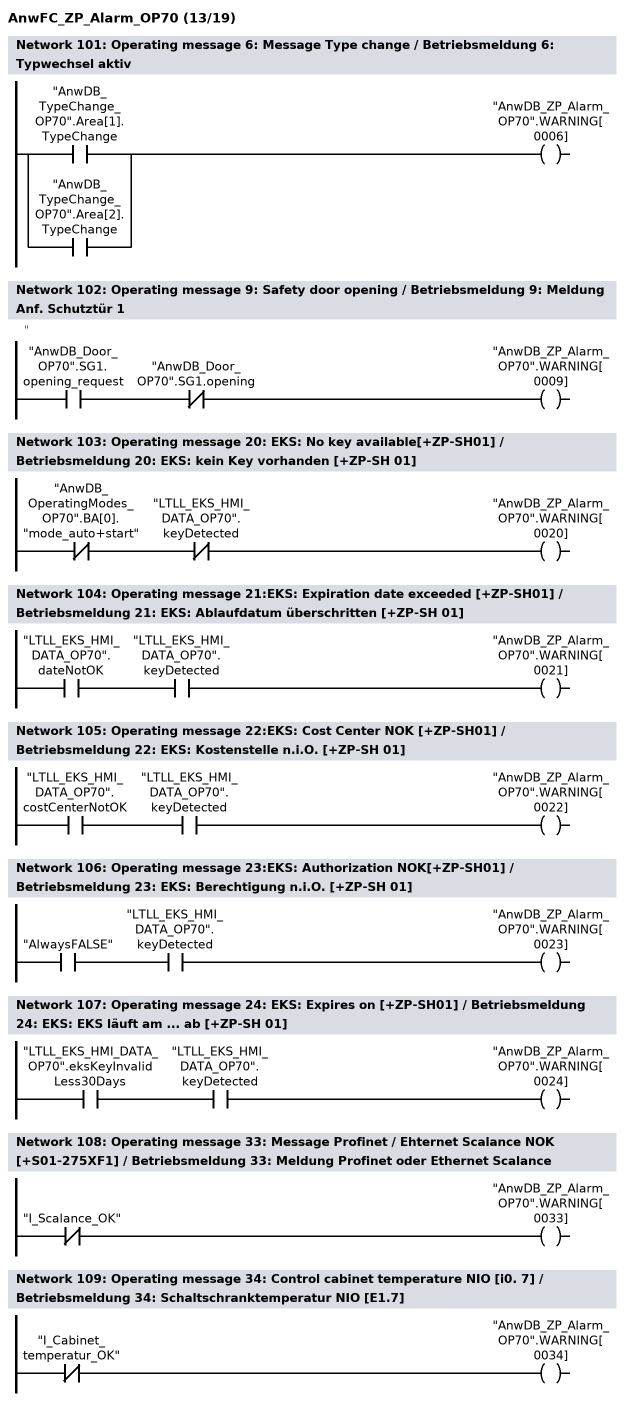
   RUNG wire#powerrail
      Contact( "AnwDB_TypeChange_OP70".Area[1].TypeChange )
      wire#w1
      Coil( "AnwDB_ZP_Alarm_OP70".WARNING[0006] )
   END_RUNG
   RUNG wire#powerrail
      Contact( "AnwDB_TypeChange_OP70".Area[2].TypeChange )
   END_RUNG wire#w1
   // the same network as SCL:
   "AnwDB_ZP_Alarm_OP70".WARNING[0006] := "AnwDB_TypeChange_OP70".Area[1].TypeChange OR "AnwDB_TypeChange_OP70".Area[2].TypeChange;
END_REGION

REGION Network 102: Operating message 9: Safety door opening / Betriebsmeldung 9: Meldung Anf. Schutztür 1
   // "
   RUNG wire#powerrail
      Contact( "AnwDB_Door_OP70".SG1.opening_request )
      I_Contact( "AnwDB_Door_OP70".SG1.opening )
      Coil( "AnwDB_ZP_Alarm_OP70".WARNING[0009] )
   END_RUNG
   // the same network as SCL:
   "AnwDB_ZP_Alarm_OP70".WARNING[0009] := "AnwDB_Door_OP70".SG1.opening_request AND NOT "AnwDB_Door_OP70".SG1.opening;
END_REGION

REGION Network 103: Operating message 20: EKS: No key available[+ZP-SH01] / Betriebsmeldung 20: EKS: kein Key vorhanden [+ZP-SH 01]
   RUNG wire#powerrail
      I_Contact( "AnwDB_OperatingModes_OP70".BA[0]."mode_auto+start" )
      I_Contact( "LTLL_EKS_HMI_DATA_OP70".keyDetected )
      Coil( "AnwDB_ZP_Alarm_OP70".WARNING[0020] )
   END_RUNG
   // the same network as SCL:
   "AnwDB_ZP_Alarm_OP70".WARNING[0020] := NOT "AnwDB_OperatingModes_OP70".BA[0]."mode_auto+start" AND NOT "LTLL_EKS_HMI_DATA_OP70".keyDetected;
END_REGION

REGION Network 104: Operating message 21:EKS: Expiration date exceeded [+ZP-SH01] / Betriebsmeldung 21: EKS: Ablaufdatum überschritten [+ZP-SH 01]
   RUNG wire#powerrail
      Contact( "LTLL_EKS_HMI_DATA_OP70".dateNotOK )
      Contact( "LTLL_EKS_HMI_DATA_OP70".keyDetected )
      Coil( "AnwDB_ZP_Alarm_OP70".WARNING[0021] )
   END_RUNG
   // the same network as SCL:
   "AnwDB_ZP_Alarm_OP70".WARNING[0021] := "LTLL_EKS_HMI_DATA_OP70".dateNotOK AND "LTLL_EKS_HMI_DATA_OP70".keyDetected;
END_REGION

REGION Network 105: Operating message 22:EKS: Cost Center NOK [+ZP-SH01] / Betriebsmeldung 22: EKS: Kostenstelle n.i.O. [+ZP-SH 01]
   RUNG wire#powerrail
      Contact( "LTLL_EKS_HMI_DATA_OP70".costCenterNotOK )
      Contact( "LTLL_EKS_HMI_DATA_OP70".keyDetected )
      Coil( "AnwDB_ZP_Alarm_OP70".WARNING[0022] )
   END_RUNG
   // the same network as SCL:
   "AnwDB_ZP_Alarm_OP70".WARNING[0022] := "LTLL_EKS_HMI_DATA_OP70".costCenterNotOK AND "LTLL_EKS_HMI_DATA_OP70".keyDetected;
END_REGION

REGION Network 106: Operating message 23:EKS: Authorization NOK[+ZP-SH01] / Betriebsmeldung 23: EKS: Berechtigung n.i.O. [+ZP-SH 01]
   RUNG wire#powerrail
      Contact( "AlwaysFALSE" )
      Contact( "LTLL_EKS_HMI_DATA_OP70".keyDetected )
      Coil( "AnwDB_ZP_Alarm_OP70".WARNING[0023] )
   END_RUNG
   // the same network as SCL:
   "AnwDB_ZP_Alarm_OP70".WARNING[0023] := "AlwaysFALSE" AND "LTLL_EKS_HMI_DATA_OP70".keyDetected;
END_REGION

REGION Network 107: Operating message 24: EKS: Expires on [+ZP-SH01] / Betriebsmeldung 24: EKS: EKS läuft am ... ab [+ZP-SH 01]
   RUNG wire#powerrail
      Contact( "LTLL_EKS_HMI_DATA_OP70".eksKeyInvalidLess30Days )
      Contact( "LTLL_EKS_HMI_DATA_OP70".keyDetected )
      Coil( "AnwDB_ZP_Alarm_OP70".WARNING[0024] )
   END_RUNG
   // the same network as SCL:
   "AnwDB_ZP_Alarm_OP70".WARNING[0024] := "LTLL_EKS_HMI_DATA_OP70".eksKeyInvalidLess30Days AND "LTLL_EKS_HMI_DATA_OP70".keyDetected;
END_REGION

REGION Network 108: Operating message 33: Message Profinet / Ehternet Scalance NOK [+S01-275XF1] / Betriebsmeldung 33: Meldung Profinet oder Ethernet Scalance
   RUNG wire#powerrail
      I_Contact( "I_Scalance_OK" )
      Coil( "AnwDB_ZP_Alarm_OP70".WARNING[0033] )
   END_RUNG
   // the same network as SCL:
   "AnwDB_ZP_Alarm_OP70".WARNING[0033] := NOT "I_Scalance_OK";
END_REGION

REGION Network 109: Operating message 34: Control cabinet temperature NIO [i0. 7] / Betriebsmeldung 34: Schaltschranktemperatur NIO [E1.7]
   RUNG wire#powerrail
      I_Contact( "I_Cabinet_temperatur_OK" )
      Coil( "AnwDB_ZP_Alarm_OP70".WARNING[0034] )
   END_RUNG
   // the same network as SCL:
   "AnwDB_ZP_Alarm_OP70".WARNING[0034] := NOT "I_Cabinet_temperatur_OK";
END_REGION

REGION Network 110: Operating message 50: Removed at least one processing. / Betriebsmeldung 50: Mindestens eine Bearbeitung abgewählt
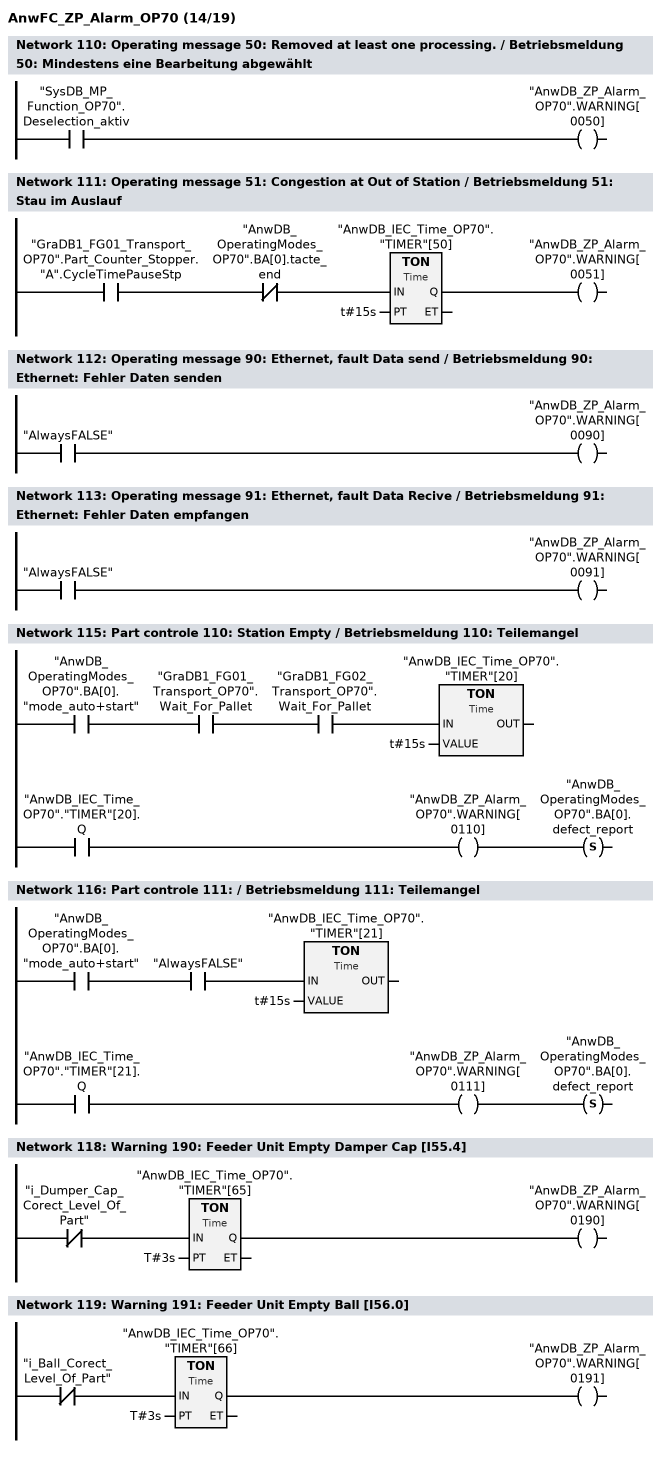
   RUNG wire#powerrail
      Contact( "SysDB_MP_Function_OP70".Deselection_aktiv )
      Coil( "AnwDB_ZP_Alarm_OP70".WARNING[0050] )
   END_RUNG
   // the same network as SCL:
   "AnwDB_ZP_Alarm_OP70".WARNING[0050] := "SysDB_MP_Function_OP70".Deselection_aktiv;
END_REGION

REGION Network 111: Operating message 51: Congestion at Out of Station / Betriebsmeldung 51: Stau im Auslauf
   RUNG wire#powerrail
      Contact( "GraDB1_FG01_Transport_OP70".Part_Counter_Stopper."A".CycleTimePauseStp )
      I_Contact( "AnwDB_OperatingModes_OP70".BA[0].tacte_end )
      { S7_Templates := "time_type := Time" } "AnwDB_IEC_Time_OP70"."TIMER"[50].TON(pt := t#15s, et =>)
      Coil( "AnwDB_ZP_Alarm_OP70".WARNING[0051] )
   END_RUNG
   // the same network as SCL:
   "AnwDB_IEC_Time_OP70"."TIMER"[50].TON(IN := "GraDB1_FG01_Transport_OP70".Part_Counter_Stopper."A".CycleTimePauseStp AND NOT "AnwDB_OperatingModes_OP70".BA[0].tacte_end,
                           PT := t#15s);
   "AnwDB_ZP_Alarm_OP70".WARNING[0051] := "AnwDB_IEC_Time_OP70"."TIMER"[50].Q;
END_REGION

REGION Network 112: Operating message 90: Ethernet, fault Data send / Betriebsmeldung 90: Ethernet: Fehler Daten senden
   RUNG wire#powerrail
      Contact( "AlwaysFALSE" )
      Coil( "AnwDB_ZP_Alarm_OP70".WARNING[0090] )
   END_RUNG
   // the same network as SCL:
   "AnwDB_ZP_Alarm_OP70".WARNING[0090] := "AlwaysFALSE";
END_REGION

REGION Network 113: Operating message 91: Ethernet, fault Data Recive / Betriebsmeldung 91: Ethernet: Fehler Daten empfangen
   RUNG wire#powerrail
      Contact( "AlwaysFALSE" )
      Coil( "AnwDB_ZP_Alarm_OP70".WARNING[0091] )
   END_RUNG
   // the same network as SCL:
   "AnwDB_ZP_Alarm_OP70".WARNING[0091] := "AlwaysFALSE";
END_REGION

REGION Network 114: #################### MANGELMELDUNG #####################
END_REGION

REGION Network 115: Part controle 110: Station Empty / Betriebsmeldung 110: Teilemangel
   "AnwDB_IEC_Time_OP70"."TIMER"[20].TON(IN := "AnwDB_OperatingModes_OP70".BA[0]."mode_auto+start" AND "GraDB1_FG01_Transport_OP70".Wait_For_Pallet AND "GraDB1_FG02_Transport_OP70".Wait_For_Pallet, PT := t#15s);   // TON coil
   "AnwDB_ZP_Alarm_OP70".WARNING[0110] := "AnwDB_IEC_Time_OP70"."TIMER"[20].Q;
   IF "AnwDB_IEC_Time_OP70"."TIMER"[20].Q THEN
       "AnwDB_OperatingModes_OP70".BA[0].defect_report := TRUE;
   END_IF;
END_REGION

REGION Network 116: Part controle 111: / Betriebsmeldung 111: Teilemangel
   "AnwDB_IEC_Time_OP70"."TIMER"[21].TON(IN := "AnwDB_OperatingModes_OP70".BA[0]."mode_auto+start" AND "AlwaysFALSE", PT := t#15s);   // TON coil
   "AnwDB_ZP_Alarm_OP70".WARNING[0111] := "AnwDB_IEC_Time_OP70"."TIMER"[21].Q;
   IF "AnwDB_IEC_Time_OP70"."TIMER"[21].Q THEN
       "AnwDB_OperatingModes_OP70".BA[0].defect_report := TRUE;
   END_IF;
END_REGION

REGION Network 117: #################### External SYSTEME ##################### / #################### SUBSYSTEME #####################
END_REGION

REGION Network 118: Warning 190: Feeder Unit Empty Damper Cap [I55.4]
   RUNG wire#powerrail
      I_Contact( "i_Dumper_Cap_Corect_Level_Of_Part" )
      { S7_Templates := "time_type := Time" } "AnwDB_IEC_Time_OP70"."TIMER"[65].TON(pt := T#3s, et =>)
      Coil( "AnwDB_ZP_Alarm_OP70".WARNING[0190] )
   END_RUNG
   // the same network as SCL:
   "AnwDB_IEC_Time_OP70"."TIMER"[65].TON(IN := NOT "i_Dumper_Cap_Corect_Level_Of_Part", PT := T#3s);
   "AnwDB_ZP_Alarm_OP70".WARNING[0190] := "AnwDB_IEC_Time_OP70"."TIMER"[65].Q;
END_REGION

REGION Network 119: Warning 191: Feeder Unit Empty Ball [I56.0]
   RUNG wire#powerrail
      I_Contact( "i_Ball_Corect_Level_Of_Part" )
      { S7_Templates := "time_type := Time" } "AnwDB_IEC_Time_OP70"."TIMER"[66].TON(pt := T#3s, et =>)
      Coil( "AnwDB_ZP_Alarm_OP70".WARNING[0191] )
   END_RUNG
   // the same network as SCL:
   "AnwDB_IEC_Time_OP70"."TIMER"[66].TON(IN := NOT "i_Ball_Corect_Level_Of_Part", PT := T#3s);
   "AnwDB_ZP_Alarm_OP70".WARNING[0191] := "AnwDB_IEC_Time_OP70"."TIMER"[66].Q;
END_REGION

REGION Network 120: Warning 192: Feeder Unit Empty Screw [I56.1]
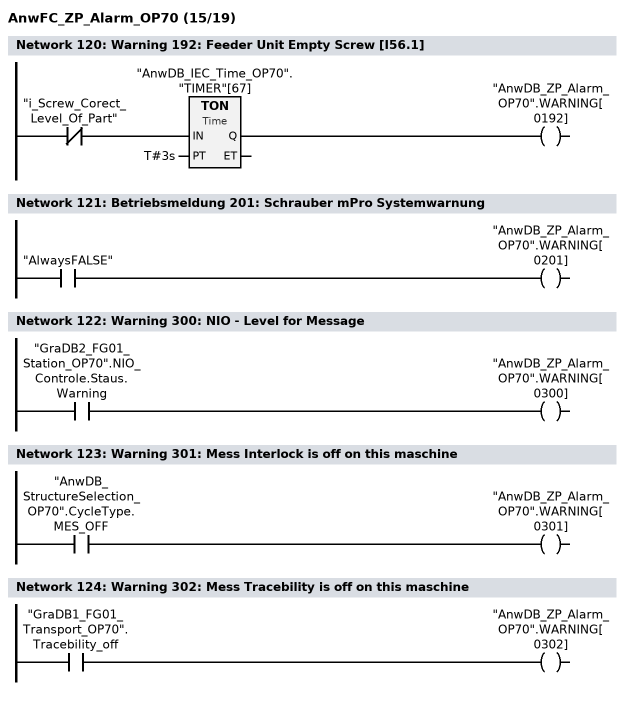
   RUNG wire#powerrail
      I_Contact( "i_Screw_Corect_Level_Of_Part" )
      { S7_Templates := "time_type := Time" } "AnwDB_IEC_Time_OP70"."TIMER"[67].TON(pt := T#3s, et =>)
      Coil( "AnwDB_ZP_Alarm_OP70".WARNING[0192] )
   END_RUNG
   // the same network as SCL:
   "AnwDB_IEC_Time_OP70"."TIMER"[67].TON(IN := NOT "i_Screw_Corect_Level_Of_Part", PT := T#3s);
   "AnwDB_ZP_Alarm_OP70".WARNING[0192] := "AnwDB_IEC_Time_OP70"."TIMER"[67].Q;
END_REGION

REGION Network 121: Betriebsmeldung 201: Schrauber mPro Systemwarnung
   RUNG wire#powerrail
      Contact( "AlwaysFALSE" )
      Coil( "AnwDB_ZP_Alarm_OP70".WARNING[0201] )
   END_RUNG
   // the same network as SCL:
   "AnwDB_ZP_Alarm_OP70".WARNING[0201] := "AlwaysFALSE";
END_REGION

REGION Network 122: Warning 300: NIO - Level for Message
   RUNG wire#powerrail
      Contact( "GraDB2_FG01_Station_OP70".NIO_Controle.Staus.Warning )
      Coil( "AnwDB_ZP_Alarm_OP70".WARNING[0300] )
   END_RUNG
   // the same network as SCL:
   "AnwDB_ZP_Alarm_OP70".WARNING[0300] := "GraDB2_FG01_Station_OP70".NIO_Controle.Staus.Warning;
END_REGION

REGION Network 123: Warning 301: Mess Interlock is off on this maschine
   RUNG wire#powerrail
      Contact( "AnwDB_StructureSelection_OP70".CycleType.MES_OFF )
      Coil( "AnwDB_ZP_Alarm_OP70".WARNING[0301] )
   END_RUNG
   // the same network as SCL:
   "AnwDB_ZP_Alarm_OP70".WARNING[0301] := "AnwDB_StructureSelection_OP70".CycleType.MES_OFF;
END_REGION

REGION Network 124: Warning 302: Mess Tracebility is off on this maschine
   RUNG wire#powerrail
      Contact( "GraDB1_FG01_Transport_OP70".Tracebility_off )
      Coil( "AnwDB_ZP_Alarm_OP70".WARNING[0302] )
   END_RUNG
   // the same network as SCL:
   "AnwDB_ZP_Alarm_OP70".WARNING[0302] := "GraDB1_FG01_Transport_OP70".Tracebility_off;
END_REGION

REGION Network 125: Warning 303: Waiting for MES response (ISynchro=2)
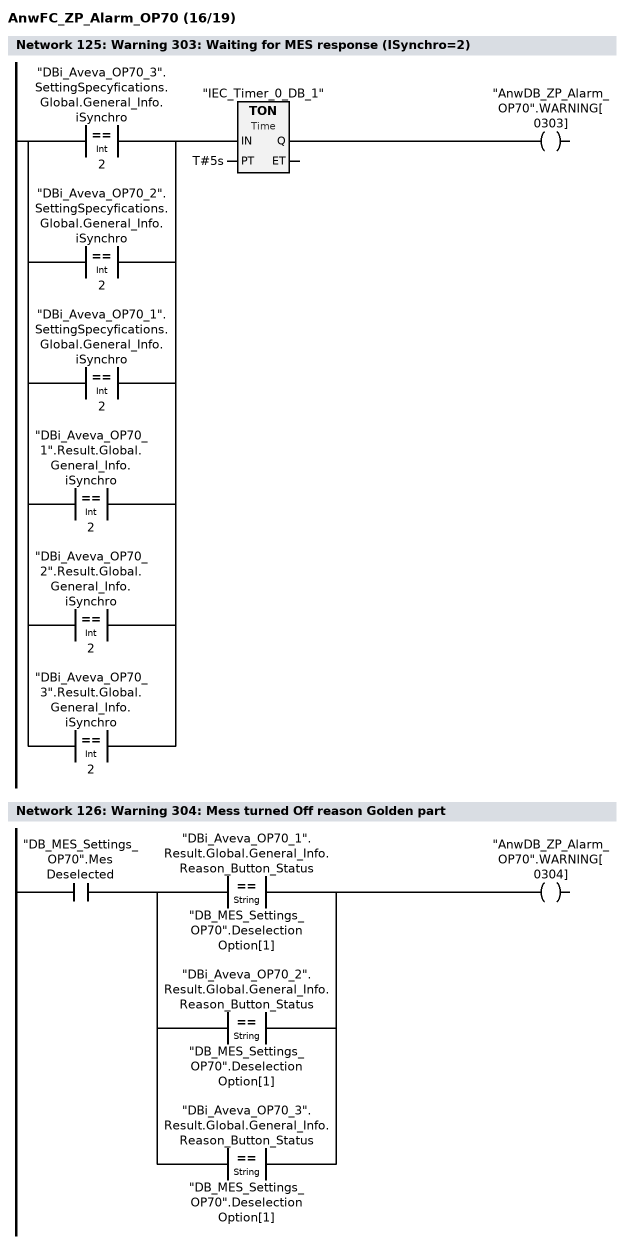
   RUNG wire#powerrail
      { S7_Templates := "SrcType := Int" } EQ_Contact(in1 := "DBi_Aveva_OP70_3".SettingSpecyfications.Global.General_Info.iSynchro, in2 := 2)
      wire#w1
      { S7_Templates := "time_type := Time" } "IEC_Timer_0_DB_1".TON(pt := T#5s, et =>)
      Coil( "AnwDB_ZP_Alarm_OP70".WARNING[0303] )
   END_RUNG
   RUNG wire#powerrail
      { S7_Templates := "SrcType := Int" } EQ_Contact(in1 := "DBi_Aveva_OP70_2".SettingSpecyfications.Global.General_Info.iSynchro, in2 := 2)
   END_RUNG wire#w1
   RUNG wire#powerrail
      { S7_Templates := "SrcType := Int" } EQ_Contact(in1 := "DBi_Aveva_OP70_1".SettingSpecyfications.Global.General_Info.iSynchro, in2 := 2)
   END_RUNG wire#w1
   RUNG wire#powerrail
      { S7_Templates := "SrcType := Int" } EQ_Contact(in1 := "DBi_Aveva_OP70_1".Result.Global.General_Info.iSynchro, in2 := 2)
   END_RUNG wire#w1
   RUNG wire#powerrail
      { S7_Templates := "SrcType := Int" } EQ_Contact(in1 := "DBi_Aveva_OP70_2".Result.Global.General_Info.iSynchro, in2 := 2)
   END_RUNG wire#w1
   RUNG wire#powerrail
      { S7_Templates := "SrcType := Int" } EQ_Contact(in1 := "DBi_Aveva_OP70_3".Result.Global.General_Info.iSynchro, in2 := 2)
   END_RUNG wire#w1
   // the same network as SCL:
   "IEC_Timer_0_DB_1".TON(IN := ("DBi_Aveva_OP70_3".SettingSpecyfications.Global.General_Info.iSynchro = 2) OR ("DBi_Aveva_OP70_2".SettingSpecyfications.Global.General_Info.iSynchro = 2) OR ("DBi_Aveva_OP70_1".SettingSpecyfications.Global.General_Info.iSynchro = 2) OR ("DBi_Aveva_OP70_1".Result.Global.General_Info.iSynchro = 2) OR ("DBi_Aveva_OP70_2".Result.Global.General_Info.iSynchro = 2) OR ("DBi_Aveva_OP70_3".Result.Global.General_Info.iSynchro = 2),
                          PT := T#5s);
   "AnwDB_ZP_Alarm_OP70".WARNING[0303] := "IEC_Timer_0_DB_1".Q;
END_REGION

REGION Network 126: Warning 304: Mess turned Off reason Golden part
   RUNG wire#powerrail
      Contact( "DB_MES_Settings_OP70".MesDeselected )
      wire#w1
      { S7_Templates := "SrcType := String" } EQ_Contact(in1 := "DBi_Aveva_OP70_1".Result.Global.General_Info.Reason_Button_Status, in2 := "DB_MES_Settings_OP70".DeselectionOption[1])
      wire#w2
      Coil( "AnwDB_ZP_Alarm_OP70".WARNING[0304] )
   END_RUNG
   RUNG wire#w1
      { S7_Templates := "SrcType := String" } EQ_Contact(in1 := "DBi_Aveva_OP70_2".Result.Global.General_Info.Reason_Button_Status, in2 := "DB_MES_Settings_OP70".DeselectionOption[1])
   END_RUNG wire#w2
   RUNG wire#w1
      { S7_Templates := "SrcType := String" } EQ_Contact(in1 := "DBi_Aveva_OP70_3".Result.Global.General_Info.Reason_Button_Status, in2 := "DB_MES_Settings_OP70".DeselectionOption[1])
   END_RUNG wire#w2
   // the same network as SCL:
   "AnwDB_ZP_Alarm_OP70".WARNING[0304] := "DB_MES_Settings_OP70".MesDeselected AND (("DBi_Aveva_OP70_1".Result.Global.General_Info.Reason_Button_Status = "DB_MES_Settings_OP70".DeselectionOption[1]) OR ("DBi_Aveva_OP70_2".Result.Global.General_Info.Reason_Button_Status = "DB_MES_Settings_OP70".DeselectionOption[1]) OR ("DBi_Aveva_OP70_3".Result.Global.General_Info.Reason_Button_Status = "DB_MES_Settings_OP70".DeselectionOption[1]));
END_REGION

REGION Network 127: Warning 305: Mess turned Off reason Maintenance
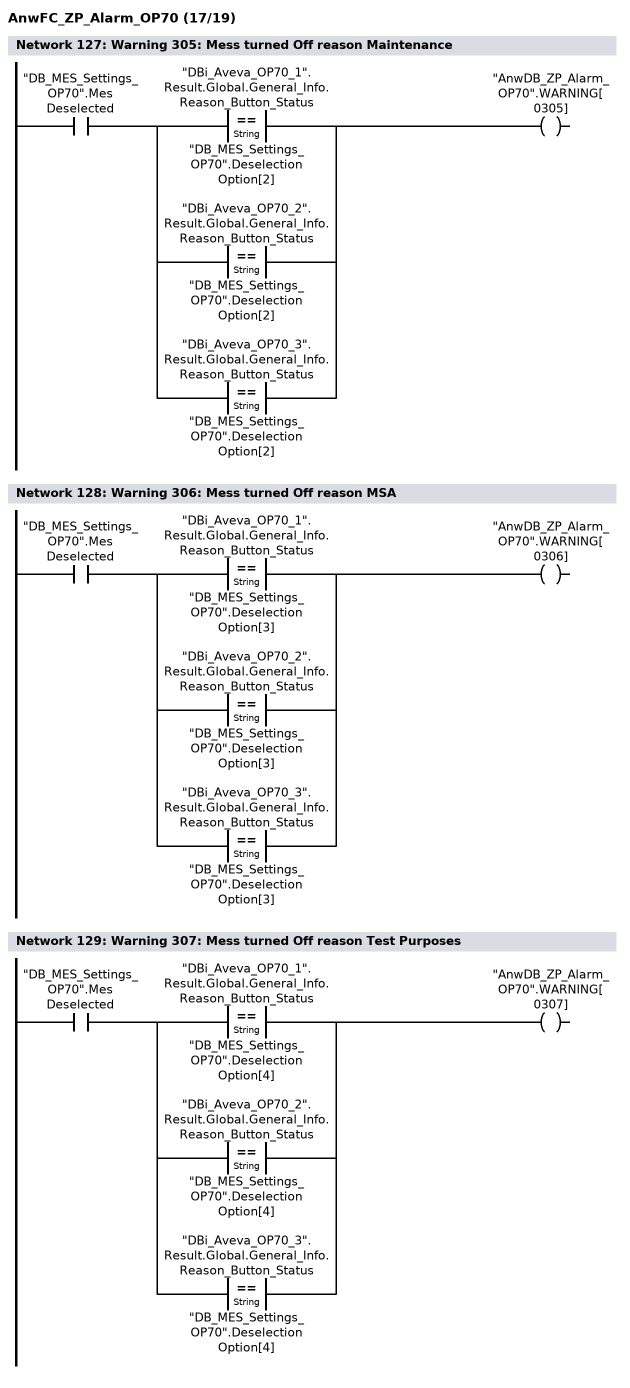
   RUNG wire#powerrail
      Contact( "DB_MES_Settings_OP70".MesDeselected )
      wire#w1
      { S7_Templates := "SrcType := String" } EQ_Contact(in1 := "DBi_Aveva_OP70_1".Result.Global.General_Info.Reason_Button_Status, in2 := "DB_MES_Settings_OP70".DeselectionOption[2])
      wire#w2
      Coil( "AnwDB_ZP_Alarm_OP70".WARNING[0305] )
   END_RUNG
   RUNG wire#w1
      { S7_Templates := "SrcType := String" } EQ_Contact(in1 := "DBi_Aveva_OP70_2".Result.Global.General_Info.Reason_Button_Status, in2 := "DB_MES_Settings_OP70".DeselectionOption[2])
   END_RUNG wire#w2
   RUNG wire#w1
      { S7_Templates := "SrcType := String" } EQ_Contact(in1 := "DBi_Aveva_OP70_3".Result.Global.General_Info.Reason_Button_Status, in2 := "DB_MES_Settings_OP70".DeselectionOption[2])
   END_RUNG wire#w2
   // the same network as SCL:
   "AnwDB_ZP_Alarm_OP70".WARNING[0305] := "DB_MES_Settings_OP70".MesDeselected AND (("DBi_Aveva_OP70_1".Result.Global.General_Info.Reason_Button_Status = "DB_MES_Settings_OP70".DeselectionOption[2]) OR ("DBi_Aveva_OP70_2".Result.Global.General_Info.Reason_Button_Status = "DB_MES_Settings_OP70".DeselectionOption[2]) OR ("DBi_Aveva_OP70_3".Result.Global.General_Info.Reason_Button_Status = "DB_MES_Settings_OP70".DeselectionOption[2]));
END_REGION

REGION Network 128: Warning 306: Mess turned Off reason MSA
   RUNG wire#powerrail
      Contact( "DB_MES_Settings_OP70".MesDeselected )
      wire#w1
      { S7_Templates := "SrcType := String" } EQ_Contact(in1 := "DBi_Aveva_OP70_1".Result.Global.General_Info.Reason_Button_Status, in2 := "DB_MES_Settings_OP70".DeselectionOption[3])
      wire#w2
      Coil( "AnwDB_ZP_Alarm_OP70".WARNING[0306] )
   END_RUNG
   RUNG wire#w1
      { S7_Templates := "SrcType := String" } EQ_Contact(in1 := "DBi_Aveva_OP70_2".Result.Global.General_Info.Reason_Button_Status, in2 := "DB_MES_Settings_OP70".DeselectionOption[3])
   END_RUNG wire#w2
   RUNG wire#w1
      { S7_Templates := "SrcType := String" } EQ_Contact(in1 := "DBi_Aveva_OP70_3".Result.Global.General_Info.Reason_Button_Status, in2 := "DB_MES_Settings_OP70".DeselectionOption[3])
   END_RUNG wire#w2
   // the same network as SCL:
   "AnwDB_ZP_Alarm_OP70".WARNING[0306] := "DB_MES_Settings_OP70".MesDeselected AND (("DBi_Aveva_OP70_1".Result.Global.General_Info.Reason_Button_Status = "DB_MES_Settings_OP70".DeselectionOption[3]) OR ("DBi_Aveva_OP70_2".Result.Global.General_Info.Reason_Button_Status = "DB_MES_Settings_OP70".DeselectionOption[3]) OR ("DBi_Aveva_OP70_3".Result.Global.General_Info.Reason_Button_Status = "DB_MES_Settings_OP70".DeselectionOption[3]));
END_REGION

REGION Network 129: Warning 307: Mess turned Off reason Test Purposes
   RUNG wire#powerrail
      Contact( "DB_MES_Settings_OP70".MesDeselected )
      wire#w1
      { S7_Templates := "SrcType := String" } EQ_Contact(in1 := "DBi_Aveva_OP70_1".Result.Global.General_Info.Reason_Button_Status, in2 := "DB_MES_Settings_OP70".DeselectionOption[4])
      wire#w2
      Coil( "AnwDB_ZP_Alarm_OP70".WARNING[0307] )
   END_RUNG
   RUNG wire#w1
      { S7_Templates := "SrcType := String" } EQ_Contact(in1 := "DBi_Aveva_OP70_2".Result.Global.General_Info.Reason_Button_Status, in2 := "DB_MES_Settings_OP70".DeselectionOption[4])
   END_RUNG wire#w2
   RUNG wire#w1
      { S7_Templates := "SrcType := String" } EQ_Contact(in1 := "DBi_Aveva_OP70_3".Result.Global.General_Info.Reason_Button_Status, in2 := "DB_MES_Settings_OP70".DeselectionOption[4])
   END_RUNG wire#w2
   // the same network as SCL:
   "AnwDB_ZP_Alarm_OP70".WARNING[0307] := "DB_MES_Settings_OP70".MesDeselected AND (("DBi_Aveva_OP70_1".Result.Global.General_Info.Reason_Button_Status = "DB_MES_Settings_OP70".DeselectionOption[4]) OR ("DBi_Aveva_OP70_2".Result.Global.General_Info.Reason_Button_Status = "DB_MES_Settings_OP70".DeselectionOption[4]) OR ("DBi_Aveva_OP70_3".Result.Global.General_Info.Reason_Button_Status = "DB_MES_Settings_OP70".DeselectionOption[4]));
END_REGION

REGION Network 130: ############# CHEKING OUT ############## / ####################### AUSWERTUNG ########################
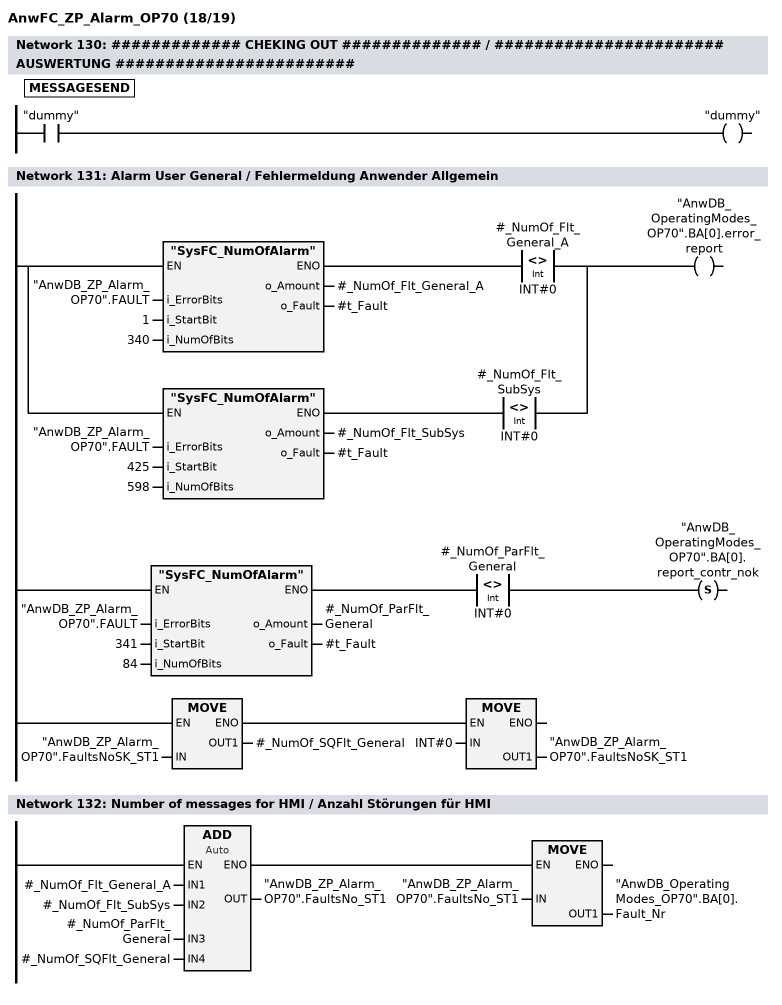
   Label( MESSAGESEND )
   RUNG wire#powerrail
      Contact( "dummy" )
      Coil( "dummy" )
   END_RUNG
   // the same network as SCL:
   MESSAGESEND:
   "dummy" := "dummy";
END_REGION

REGION Network 131: Alarm User General / Fehlermeldung Anwender Allgemein
   RUNG wire#powerrail
      "SysFC_NumOfAlarm"(i_ErrorBits := "AnwDB_ZP_Alarm_OP70".FAULT, i_StartBit := 1, i_NumOfBits := 340, o_Amount => #_NumOf_Flt_General_A, o_Fault => #t_Fault)
      { S7_Templates := "SrcType := Int" } NE_Contact(in1 := #_NumOf_Flt_General_A, in2 := INT#0)
      wire#w1
      Coil( "AnwDB_OperatingModes_OP70".BA[0].error_report )
   END_RUNG
   RUNG wire#powerrail
      "SysFC_NumOfAlarm"(i_ErrorBits := "AnwDB_ZP_Alarm_OP70".FAULT, i_StartBit := 425, i_NumOfBits := 598, o_Amount => #_NumOf_Flt_SubSys, o_Fault => #t_Fault)
      { S7_Templates := "SrcType := Int" } NE_Contact(in1 := #_NumOf_Flt_SubSys, in2 := INT#0)
   END_RUNG wire#w1
   RUNG wire#powerrail
      "SysFC_NumOfAlarm"(i_ErrorBits := "AnwDB_ZP_Alarm_OP70".FAULT, i_StartBit := 341, i_NumOfBits := 84, o_Amount => #_NumOf_ParFlt_General, o_Fault => #t_Fault)
      { S7_Templates := "SrcType := Int" } NE_Contact(in1 := #_NumOf_ParFlt_General, in2 := INT#0)
      S_Coil( "AnwDB_OperatingModes_OP70".BA[0].report_contr_nok )
   END_RUNG
   RUNG wire#powerrail
      { S7_GenerateENO := "TRUE" } Move(in := "AnwDB_ZP_Alarm_OP70".FaultsNoSK_ST1, out1 => #_NumOf_SQFlt_General)
      { S7_GenerateENO := "TRUE" } Move(in := INT#0, out1 => "AnwDB_ZP_Alarm_OP70".FaultsNoSK_ST1)
   END_RUNG
   // the same network as SCL:
   // ENO of a box is taken as its EN; it also drops when the box reports an error
   "SysFC_NumOfAlarm"(i_ErrorBits := "AnwDB_ZP_Alarm_OP70".FAULT,
                      i_StartBit := 1,
                      i_NumOfBits := 340,
                      o_Amount => #_NumOf_Flt_General_A,
                      o_Fault => #t_Fault,
                      ENO => #_w1);
   "SysFC_NumOfAlarm"(i_ErrorBits := "AnwDB_ZP_Alarm_OP70".FAULT,
                      i_StartBit := 425,
                      i_NumOfBits := 598,
                      o_Amount => #_NumOf_Flt_SubSys,
                      o_Fault => #t_Fault,
                      ENO => #_w2);
   "AnwDB_OperatingModes_OP70".BA[0].error_report := (#_w1 AND (#_NumOf_Flt_General_A <> INT#0)) OR (#_w2 AND (#_NumOf_Flt_SubSys <> INT#0));
   "SysFC_NumOfAlarm"(i_ErrorBits := "AnwDB_ZP_Alarm_OP70".FAULT,
                      i_StartBit := 341,
                      i_NumOfBits := 84,
                      o_Amount => #_NumOf_ParFlt_General,
                      o_Fault => #t_Fault,
                      ENO => #_w3);
   IF #_w3 AND (#_NumOf_ParFlt_General <> INT#0) THEN
       "AnwDB_OperatingModes_OP70".BA[0].report_contr_nok := TRUE;
   END_IF;
   #_NumOf_SQFlt_General := "AnwDB_ZP_Alarm_OP70".FaultsNoSK_ST1;
   "AnwDB_ZP_Alarm_OP70".FaultsNoSK_ST1 := INT#0;
END_REGION

REGION Network 132: Number of messages for HMI / Anzahl Störungen für HMI
   RUNG wire#powerrail
      Add(in1 := #_NumOf_Flt_General_A, in2 := #_NumOf_Flt_SubSys, in3 := #_NumOf_ParFlt_General, in4 := #_NumOf_SQFlt_General, out => "AnwDB_ZP_Alarm_OP70".FaultsNo_ST1)
      Move(in := "AnwDB_ZP_Alarm_OP70".FaultsNo_ST1, out1 => "AnwDB_OperatingModes_OP70".BA[0].Fault_Nr)
   END_RUNG
   // the same network as SCL:
   "AnwDB_ZP_Alarm_OP70".FaultsNo_ST1 := #_NumOf_Flt_General_A + #_NumOf_Flt_SubSys + #_NumOf_ParFlt_General + #_NumOf_SQFlt_General;
   "AnwDB_OperatingModes_OP70".BA[0].Fault_Nr := "AnwDB_ZP_Alarm_OP70".FaultsNo_ST1;
END_REGION

REGION Network 133: Alarm Station / Fehlermeldung Station
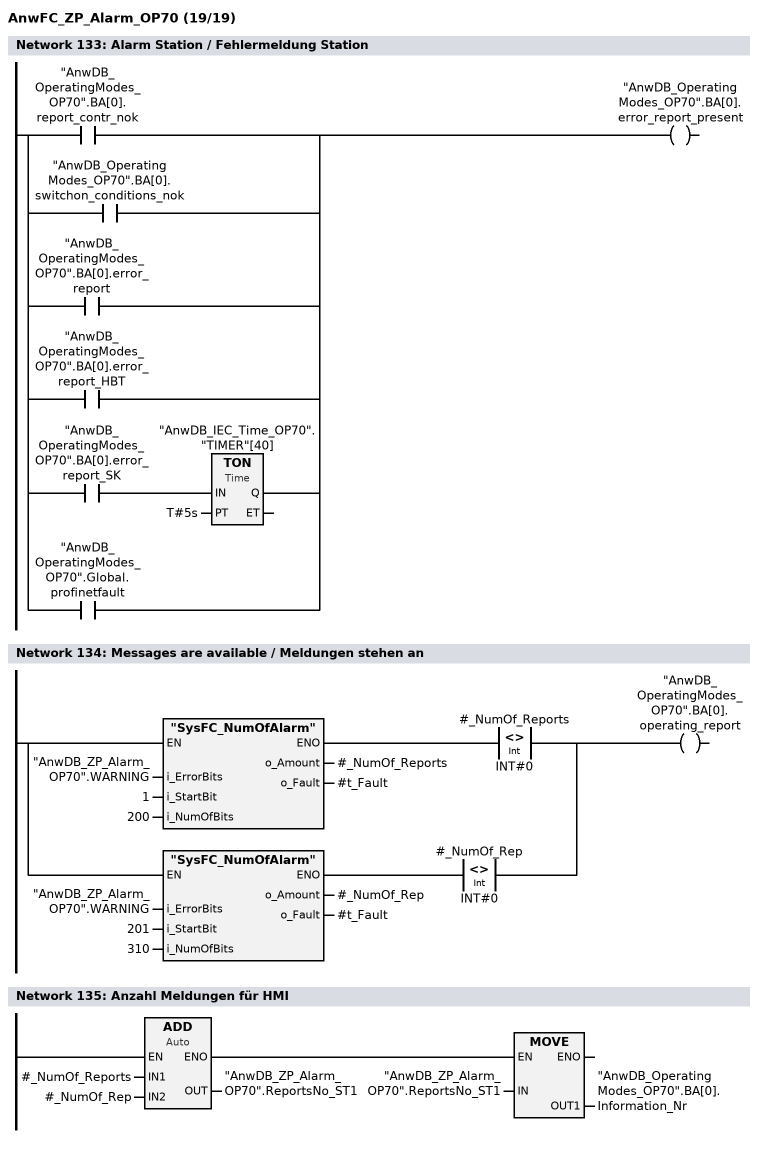
   RUNG wire#powerrail
      Contact( "AnwDB_OperatingModes_OP70".BA[0].report_contr_nok )
      wire#w1
      Coil( "AnwDB_OperatingModes_OP70".BA[0].error_report_present )
   END_RUNG
   RUNG wire#powerrail
      Contact( "AnwDB_OperatingModes_OP70".BA[0].switchon_conditions_nok )
   END_RUNG wire#w1
   RUNG wire#powerrail
      Contact( "AnwDB_OperatingModes_OP70".BA[0].error_report )
   END_RUNG wire#w1
   RUNG wire#powerrail
      Contact( "AnwDB_OperatingModes_OP70".BA[0].error_report_HBT )
   END_RUNG wire#w1
   RUNG wire#powerrail
      Contact( "AnwDB_OperatingModes_OP70".BA[0].error_report_SK )
      { S7_Templates := "time_type := Time" } "AnwDB_IEC_Time_OP70"."TIMER"[40].TON(pt := T#5s, et =>)
   END_RUNG wire#w1
   RUNG wire#powerrail
      Contact( "AnwDB_OperatingModes_OP70".Global.profinetfault )
   END_RUNG wire#w1
   // the same network as SCL:
   "AnwDB_IEC_Time_OP70"."TIMER"[40].TON(IN := "AnwDB_OperatingModes_OP70".BA[0].error_report_SK, PT := T#5s);
   "AnwDB_OperatingModes_OP70".BA[0].error_report_present := "AnwDB_OperatingModes_OP70".BA[0].report_contr_nok OR "AnwDB_OperatingModes_OP70".BA[0].switchon_conditions_nok OR "AnwDB_OperatingModes_OP70".BA[0].error_report OR "AnwDB_OperatingModes_OP70".BA[0].error_report_HBT OR "AnwDB_IEC_Time_OP70"."TIMER"[40].Q OR "AnwDB_OperatingModes_OP70".Global.profinetfault;
END_REGION

REGION Network 134: Messages are available / Meldungen stehen an
   RUNG wire#powerrail
      "SysFC_NumOfAlarm"(i_ErrorBits := "AnwDB_ZP_Alarm_OP70".WARNING, i_StartBit := 1, i_NumOfBits := 200, o_Amount => #_NumOf_Reports, o_Fault => #t_Fault)
      { S7_Templates := "SrcType := Int" } NE_Contact(in1 := #_NumOf_Reports, in2 := INT#0)
      wire#w1
      Coil( "AnwDB_OperatingModes_OP70".BA[0].operating_report )
   END_RUNG
   RUNG wire#powerrail
      "SysFC_NumOfAlarm"(i_ErrorBits := "AnwDB_ZP_Alarm_OP70".WARNING, i_StartBit := 201, i_NumOfBits := 310, o_Amount => #_NumOf_Rep, o_Fault => #t_Fault)
      { S7_Templates := "SrcType := Int" } NE_Contact(in1 := #_NumOf_Rep, in2 := INT#0)
   END_RUNG wire#w1
   // the same network as SCL:
   "SysFC_NumOfAlarm"(i_ErrorBits := "AnwDB_ZP_Alarm_OP70".WARNING,
                      i_StartBit := 1,
                      i_NumOfBits := 200,
                      o_Amount => #_NumOf_Reports,
                      o_Fault => #t_Fault,
                      ENO => #_w1);
   "SysFC_NumOfAlarm"(i_ErrorBits := "AnwDB_ZP_Alarm_OP70".WARNING,
                      i_StartBit := 201,
                      i_NumOfBits := 310,
                      o_Amount => #_NumOf_Rep,
                      o_Fault => #t_Fault,
                      ENO => #_w2);
   "AnwDB_OperatingModes_OP70".BA[0].operating_report := (#_w1 AND (#_NumOf_Reports <> INT#0)) OR (#_w2 AND (#_NumOf_Rep <> INT#0));
END_REGION

REGION Network 135: Anzahl Meldungen für HMI
   RUNG wire#powerrail
      Add(in1 := #_NumOf_Reports, in2 := #_NumOf_Rep, out => "AnwDB_ZP_Alarm_OP70".ReportsNo_ST1)
      Move(in := "AnwDB_ZP_Alarm_OP70".ReportsNo_ST1, out1 => "AnwDB_OperatingModes_OP70".BA[0].Information_Nr)
   END_RUNG
   // the same network as SCL:
   "AnwDB_ZP_Alarm_OP70".ReportsNo_ST1 := #_NumOf_Reports + #_NumOf_Rep;
   "AnwDB_OperatingModes_OP70".BA[0].Information_Nr := "AnwDB_ZP_Alarm_OP70".ReportsNo_ST1;
END_REGION
END_FUNCTION
